//     Drive/Inputs/In/nDataIn1 <-> Inputs/Following error actual value
//     Drive/Inputs/In/nDcOutputTime <-> InfoData/DcOutputShift
//     Drive/Inputs/In/nState1 <-> Inputs/Statusword
//     Drive/Inputs/In/nState2 <-> Inputs/Statusword @bit 8
//     Drive/Inputs/In/nState4 @bit 1 <-> WcState/InputToggle
//     Drive/Inputs/In/nState4 <-> WcState/WcState
//     Drive/Outputs/Out/nCtrl1 <-> Outputs/Controlword
//     Drive/Outputs/Out/nCtrl2 <-> Outputs/Controlword @bit 8
//     Drive/Outputs/Out/nDataOut1 <-> Outputs/Target position
//     Enc/Inputs/In/nDataIn1 <-> Inputs/Position actual value
//     Enc/Inputs/In/nDataIn3 <-> Inputs/Touch probe pos1 pos value
//     Enc/Inputs/In/nDataIn5 <-> Inputs/Touch probe pos2 pos value
//     Enc/Inputs/In/nDcInputTime <-> InfoData/DcInputShift
//     Enc/Inputs/In/nState4 @bit 1 <-> WcState/InputToggle
//     Enc/Inputs/In/nState4 <-> WcState/WcState
//     Enc/Inputs/In/nState5 <-> Inputs/Touch probe status
//     Enc/Inputs/In/nState6 <-> Inputs/Touch probe status @bit 8
//     Enc/Outputs/Out/nCtrl5 <-> Outputs/Touch probe function
//     Enc/Outputs/Out/nCtrl6 <-> Outputs/Touch probe function @bit 8
//   NC-Task 1 SAF/Axes/Axis017_17 P1An_NGPush2 <-> Device 3 (EtherCAT)/Box 2 (CU1128)/正极踢单张废料(InoSV660N)
//     Drive/Inputs/In/nDataIn1 <-> Inputs/Following error actual value
//     Drive/Inputs/In/nDcOutputTime <-> InfoData/DcOutputShift
//     Drive/Inputs/In/nState1 <-> Inputs/Statusword
//     Drive/Inputs/In/nState2 <-> Inputs/Statusword @bit 8
//     Drive/Inputs/In/nState4 @bit 1 <-> WcState/InputToggle
//     Drive/Inputs/In/nState4 <-> WcState/WcState
//     Drive/Outputs/Out/nCtrl1 <-> Outputs/Controlword
//     Drive/Outputs/Out/nCtrl2 <-> Outputs/Controlword @bit 8
//     Drive/Outputs/Out/nDataOut1 <-> Outputs/Target position
//     Enc/Inputs/In/nDataIn1 <-> Inputs/Position actual value
//     Enc/Inputs/In/nDataIn3 <-> Inputs/Touch probe pos1 pos value
//     Enc/Inputs/In/nDataIn5 <-> Inputs/Touch probe pos2 pos value
//     Enc/Inputs/In/nDcInputTime <-> InfoData/DcInputShift
//     Enc/Inputs/In/nState4 @bit 1 <-> WcState/InputToggle
//     Enc/Inputs/In/nState4 <-> WcState/WcState
//     Enc/Inputs/In/nState5 <-> Inputs/Touch probe status
//     Enc/Inputs/In/nState6 <-> Inputs/Touch probe status @bit 8
//     Enc/Outputs/Out/nCtrl5 <-> Outputs/Touch probe function
//     Enc/Outputs/Out/nCtrl6 <-> Outputs/Touch probe function @bit 8
//   NC-Task 1 SAF/Axes/Axis018_18 P1An_DedustBelt <-> Device 3 (EtherCAT)/Box 2 (CU1128)/正极上表面除尘皮带(InoSV660N)
//     Drive/Inputs/In/nDataIn1 <-> Inputs/Following error actual value
//     Drive/Inputs/In/nDcOutputTime <-> InfoData/DcOutputShift
//     Drive/Inputs/In/nState1 <-> Inputs/Statusword
//     Drive/Inputs/In/nState2 <-> Inputs/Statusword @bit 8
//     Drive/Inputs/In/nState4 @bit 1 <-> WcState/InputToggle
//     Drive/Inputs/In/nState4 <-> WcState/WcState
//     Drive/Outputs/Out/nCtrl1 <-> Outputs/Controlword
//     Drive/Outputs/Out/nCtrl2 <-> Outputs/Controlword @bit 8
//     Drive/Outputs/Out/nDataOut1 <-> Outputs/Target position
//     Enc/Inputs/In/nDataIn1 <-> Inputs/Position actual value
//     Enc/Inputs/In/nDataIn3 <-> Inputs/Touch probe pos1 pos value
//     Enc/Inputs/In/nDataIn5 <-> Inputs/Touch probe pos2 pos value
//     Enc/Inputs/In/nDcInputTime <-> InfoData/DcInputShift
//     Enc/Inputs/In/nState4 @bit 1 <-> WcState/InputToggle
//     Enc/Inputs/In/nState4 <-> WcState/WcState
//     Enc/Inputs/In/nState5 <-> Inputs/Touch probe status
//     Enc/Inputs/In/nState6 <-> Inputs/Touch probe status @bit 8
//     Enc/Outputs/Out/nCtrl5 <-> Outputs/Touch probe function
//     Enc/Outputs/Out/nCtrl6 <-> Outputs/Touch probe function @bit 8
//   NC-Task 1 SAF/Axes/Axis019_19 P1An_DedustReverseBelt <-> Device 3 (EtherCAT)/Box 2 (CU1128)/正极下表面除尘倒装皮带(InoSV660N)
//     Drive/Inputs/In/nDataIn1 <-> Inputs/Following error actual value
//     Drive/Inputs/In/nDcOutputTime <-> InfoData/DcOutputShift
//     Drive/Inputs/In/nState1 <-> Inputs/Statusword
//     Drive/Inputs/In/nState2 <-> Inputs/Statusword @bit 8
//     Drive/Inputs/In/nState4 @bit 1 <-> WcState/InputToggle
//     Drive/Inputs/In/nState4 <-> WcState/WcState
//     Drive/Outputs/Out/nCtrl1 <-> Outputs/Controlword
//     Drive/Outputs/Out/nCtrl2 <-> Outputs/Controlword @bit 8
//     Drive/Outputs/Out/nDataOut1 <-> Outputs/Target position
//     Enc/Inputs/In/nDataIn1 <-> Inputs/Position actual value
//     Enc/Inputs/In/nDataIn3 <-> Inputs/Touch probe pos1 pos value
//     Enc/Inputs/In/nDataIn5 <-> Inputs/Touch probe pos2 pos value
//     Enc/Inputs/In/nDcInputTime <-> InfoData/DcInputShift
//     Enc/Inputs/In/nState4 @bit 1 <-> WcState/InputToggle
//     Enc/Inputs/In/nState4 <-> WcState/WcState
//     Enc/Inputs/In/nState5 <-> Inputs/Touch probe status
//     Enc/Inputs/In/nState6 <-> Inputs/Touch probe status @bit 8
//     Enc/Outputs/Out/nCtrl5 <-> Outputs/Touch probe function
//     Enc/Outputs/Out/nCtrl6 <-> Outputs/Touch probe function @bit 8
//   NC-Task 1 SAF/Axes/Axis020_20 P1An_SubBelt1 <-> Device 3 (EtherCAT)/P2M1正极送料分段皮带1[20(模切)] (InoSV660N)
//     Drive/Inputs/In/nDataIn1 <-> Inputs/Following error actual value
//     Drive/Inputs/In/nDcOutputTime <-> InfoData/DcOutputShift
//     Drive/Inputs/In/nState1 <-> Inputs/Statusword
//     Drive/Inputs/In/nState2 <-> Inputs/Statusword @bit 8
//     Drive/Inputs/In/nState4 @bit 1 <-> WcState/InputToggle
//     Drive/Inputs/In/nState4 <-> WcState/WcState
//     Drive/Outputs/Out/nCtrl1 <-> Outputs/Controlword
//     Drive/Outputs/Out/nCtrl2 <-> Outputs/Controlword @bit 8
//     Drive/Outputs/Out/nDataOut1 <-> Outputs/Target position
//     Enc/Inputs/In/nDataIn1 <-> Inputs/Position actual value
//     Enc/Inputs/In/nDataIn3 <-> Inputs/Touch probe pos1 pos value
//     Enc/Inputs/In/nDataIn5 <-> Inputs/Touch probe pos2 pos value
//     Enc/Inputs/In/nDcInputTime <-> InfoData/DcInputShift
//     Enc/Inputs/In/nState4 @bit 1 <-> WcState/InputToggle
//     Enc/Inputs/In/nState4 <-> WcState/WcState
//     Enc/Inputs/In/nState5 <-> Inputs/Touch probe status
//     Enc/Inputs/In/nState6 <-> Inputs/Touch probe status @bit 8
//     Enc/Outputs/Out/nCtrl5 <-> Outputs/Touch probe function
//     Enc/Outputs/Out/nCtrl6 <-> Outputs/Touch probe function @bit 8
//   NC-Task 1 SAF/Axes/Axis021_21 P1An_SubBelt2 <-> Device 3 (EtherCAT)/Box 2 (CU1128)/Term 44 (CU1128-C)/P2M2正极送料分段皮带2[21(模切)] (InoSV660N)
//     Drive/Inputs/In/nDataIn1 <-> Inputs/Following error actual value
//     Drive/Inputs/In/nDcOutputTime <-> InfoData/DcOutputShift
//     Drive/Inputs/In/nState1 <-> Inputs/Statusword
//     Drive/Inputs/In/nState2 <-> Inputs/Statusword @bit 8
//     Drive/Inputs/In/nState4 @bit 1 <-> WcState/InputToggle
//     Drive/Inputs/In/nState4 <-> WcState/WcState
//     Drive/Outputs/Out/nCtrl1 <-> Outputs/Controlword
//     Drive/Outputs/Out/nCtrl2 <-> Outputs/Controlword @bit 8
//     Drive/Outputs/Out/nDataOut1 <-> Outputs/Target position
//     Enc/Inputs/In/nDataIn1 <-> Inputs/Position actual value
//     Enc/Inputs/In/nDataIn3 <-> Inputs/Touch probe pos1 pos value
//     Enc/Inputs/In/nDataIn5 <-> Inputs/Touch probe pos2 pos value
//     Enc/Inputs/In/nDcInputTime <-> InfoData/DcInputShift
//     Enc/Inputs/In/nState4 @bit 1 <-> WcState/InputToggle
//     Enc/Inputs/In/nState4 <-> WcState/WcState
//     Enc/Inputs/In/nState5 <-> Inputs/Touch probe status
//     Enc/Inputs/In/nState6 <-> Inputs/Touch probe status @bit 8
//     Enc/Outputs/Out/nCtrl5 <-> Outputs/Touch probe function
//     Enc/Outputs/Out/nCtrl6 <-> Outputs/Touch probe function @bit 8
//   NC-Task 1 SAF/Axes/Axis022_22 P1An_SubBelt3 <-> Device 3 (EtherCAT)/Box 2 (CU1128)/Term 44 (CU1128-C)/P2M3正极送料分段皮带3（22模切） (InoSV660N)
//     Drive/Inputs/In/nDataIn1 <-> Inputs/Following error actual value
//     Drive/Inputs/In/nDcOutputTime <-> InfoData/DcOutputShift
//     Drive/Inputs/In/nState1 <-> Inputs/Statusword
//     Drive/Inputs/In/nState2 <-> Inputs/Statusword @bit 8
//     Drive/Inputs/In/nState4 @bit 1 <-> WcState/InputToggle
//     Drive/Inputs/In/nState4 <-> WcState/WcState
//     Drive/Outputs/Out/nCtrl1 <-> Outputs/Controlword
//     Drive/Outputs/Out/nCtrl2 <-> Outputs/Controlword @bit 8
//     Drive/Outputs/Out/nDataOut1 <-> Outputs/Target position
//     Enc/Inputs/In/nDataIn1 <-> Inputs/Position actual value
//     Enc/Inputs/In/nDataIn3 <-> Inputs/Touch probe pos1 pos value
//     Enc/Inputs/In/nDataIn5 <-> Inputs/Touch probe pos2 pos value
//     Enc/Inputs/In/nDcInputTime <-> InfoData/DcInputShift
//     Enc/Inputs/In/nState4 @bit 1 <-> WcState/InputToggle
//     Enc/Inputs/In/nState4 <-> WcState/WcState
//     Enc/Inputs/In/nState5 <-> Inputs/Touch probe status
//     Enc/Inputs/In/nState6 <-> Inputs/Touch probe status @bit 8
//     Enc/Outputs/Out/nCtrl5 <-> Outputs/Touch probe function
//     Enc/Outputs/Out/nCtrl6 <-> Outputs/Touch probe function @bit 8
//   NC-Task 1 SAF/Axes/Axis025_25 P1Ca_UnWind_L <-> Device 3 (EtherCAT)/Box 2 (CU1128)/Term 24 (CU1128-B)/负极左放卷电机(InoSV660N)
//     Drive/Inputs/In/nDataIn1 <-> Inputs/Following error actual value
//     Drive/Inputs/In/nDcOutputTime <-> InfoData/DcOutputShift
//     Drive/Inputs/In/nState1 <-> Inputs/Statusword
//     Drive/Inputs/In/nState2 <-> Inputs/Statusword @bit 8
//     Drive/Inputs/In/nState4 @bit 1 <-> WcState/InputToggle
//     Drive/Inputs/In/nState4 <-> WcState/WcState
//     Drive/Outputs/Out/nCtrl1 <-> Outputs/Controlword
//     Drive/Outputs/Out/nCtrl2 <-> Outputs/Controlword @bit 8
//     Drive/Outputs/Out/nDataOut1 <-> Outputs/Target position
//     Enc/Inputs/In/nDataIn1 <-> Inputs/Position actual value
//     Enc/Inputs/In/nDataIn3 <-> Inputs/Touch probe pos1 pos value
//     Enc/Inputs/In/nDataIn5 <-> Inputs/Touch probe pos2 pos value
//     Enc/Inputs/In/nDcInputTime <-> InfoData/DcInputShift
//     Enc/Inputs/In/nState4 @bit 1 <-> WcState/InputToggle
//     Enc/Inputs/In/nState4 <-> WcState/WcState
//     Enc/Inputs/In/nState5 <-> Inputs/Touch probe status
//     Enc/Inputs/In/nState6 <-> Inputs/Touch probe status @bit 8
//     Enc/Outputs/Out/nCtrl5 <-> Outputs/Touch probe function
//     Enc/Outputs/Out/nCtrl6 <-> Outputs/Touch probe function @bit 8
//   NC-Task 1 SAF/Axes/Axis026_26 P1Ca_UnWind_R <-> Device 3 (EtherCAT)/Box 2 (CU1128)/Term 24 (CU1128-B)/负极右放卷电机(InoSV660N)
//     Drive/Inputs/In/nDataIn1 <-> Inputs/Following error actual value
//     Drive/Inputs/In/nDcOutputTime <-> InfoData/DcOutputShift
//     Drive/Inputs/In/nState1 <-> Inputs/Statusword
//     Drive/Inputs/In/nState2 <-> Inputs/Statusword @bit 8
//     Drive/Inputs/In/nState4 @bit 1 <-> WcState/InputToggle
//     Drive/Inputs/In/nState4 <-> WcState/WcState
//     Drive/Outputs/Out/nCtrl1 <-> Outputs/Controlword
//     Drive/Outputs/Out/nCtrl2 <-> Outputs/Controlword @bit 8
//     Drive/Outputs/Out/nDataOut1 <-> Outputs/Target position
//     Enc/Inputs/In/nDataIn1 <-> Inputs/Position actual value
//     Enc/Inputs/In/nDataIn3 <-> Inputs/Touch probe pos1 pos value
//     Enc/Inputs/In/nDataIn5 <-> Inputs/Touch probe pos2 pos value
//     Enc/Inputs/In/nDcInputTime <-> InfoData/DcInputShift
//     Enc/Inputs/In/nState4 @bit 1 <-> WcState/InputToggle
//     Enc/Inputs/In/nState4 <-> WcState/WcState
//     Enc/Inputs/In/nState5 <-> Inputs/Touch probe status
//     Enc/Inputs/In/nState6 <-> Inputs/Touch probe status @bit 8
//     Enc/Outputs/Out/nCtrl5 <-> Outputs/Touch probe function
//     Enc/Outputs/Out/nCtrl6 <-> Outputs/Touch probe function @bit 8
//   NC-Task 1 SAF/Axes/Axis027_27 P1Ca_PoleTension <-> Device 3 (EtherCAT)/Box 2 (CU1128)/Term 24 (CU1128-B)/负极模切前摆杆张力(InoSV660N)
//     Drive/Inputs/In/nDcOutputTime <-> InfoData/DcOutputShift
//     Drive/Inputs/In/nState1 <-> Inputs/Statusword
//     Drive/Inputs/In/nState2 <-> Inputs/Statusword @bit 8
//     Drive/Inputs/In/nState4 @bit 1 <-> WcState/InputToggle
//     Drive/Inputs/In/nState4 <-> WcState/WcState
//     Drive/Inputs/In/nState5 <-> Inputs/Modes of operation display
//     Drive/Outputs/Out/nCtrl1 <-> Outputs/Controlword
//     Drive/Outputs/Out/nCtrl2 <-> Outputs/Controlword @bit 8
//     Drive/Outputs/Out/nDataOut1 <-> Outputs/Target position
//     Drive/Outputs/Out/nDataOut2 <-> Outputs/Target velocity
//     Enc/Inputs/In/nDataIn1 <-> Inputs/Position actual value
//     Enc/Inputs/In/nDataIn3 <-> Inputs/Touch probe pos1 pos value
//     Enc/Inputs/In/nDataIn5 <-> Inputs/Touch probe pos2 pos value
//     Enc/Inputs/In/nDcInputTime <-> InfoData/DcInputShift
//     Enc/Inputs/In/nState4 @bit 1 <-> WcState/InputToggle
//     Enc/Inputs/In/nState4 <-> WcState/WcState
//     Enc/Inputs/In/nState5 <-> Inputs/Touch probe status
//     Enc/Inputs/In/nState6 <-> Inputs/Touch probe status @bit 8
//     Enc/Outputs/Out/nCtrl5 <-> Outputs/Touch probe function
//     Enc/Outputs/Out/nCtrl6 <-> Outputs/Touch probe function @bit 8
//   NC-Task 1 SAF/Axes/Axis028_28 P1Ca_DriverAux <-> Device 3 (EtherCAT)/Box 2 (CU1128)/Term 24 (CU1128-B)/负极模切辅助驱动(InoSV660N)
//     Drive/Inputs/In/nDataIn1 <-> Inputs/Following error actual value
//     Drive/Inputs/In/nDcOutputTime <-> InfoData/DcOutputShift
//     Drive/Inputs/In/nState1 <-> Inputs/Statusword
//     Drive/Inputs/In/nState2 <-> Inputs/Statusword @bit 8
//     Drive/Inputs/In/nState4 @bit 1 <-> WcState/InputToggle
//     Drive/Inputs/In/nState4 <-> WcState/WcState
//     Drive/Outputs/Out/nCtrl1 <-> Outputs/Controlword
//     Drive/Outputs/Out/nCtrl2 <-> Outputs/Controlword @bit 8
//     Drive/Outputs/Out/nDataOut1 <-> Outputs/Target position
//     Enc/Inputs/In/nDataIn1 <-> Inputs/Position actual value
//     Enc/Inputs/In/nDataIn3 <-> Inputs/Touch probe pos1 pos value
//     Enc/Inputs/In/nDataIn5 <-> Inputs/Touch probe pos2 pos value
//     Enc/Inputs/In/nDcInputTime <-> InfoData/DcInputShift
//     Enc/Inputs/In/nState4 @bit 1 <-> WcState/InputToggle
//     Enc/Inputs/In/nState4 <-> WcState/WcState
//     Enc/Inputs/In/nState5 <-> Inputs/Touch probe status
//     Enc/Inputs/In/nState6 <-> Inputs/Touch probe status @bit 8
//     Enc/Outputs/Out/nCtrl5 <-> Outputs/Touch probe function
//     Enc/Outputs/Out/nCtrl6 <-> Outputs/Touch probe function @bit 8
//   NC-Task 1 SAF/Axes/Axis029_29 P1Ca_BuffeLine <-> Device 3 (EtherCAT)/Box 2 (CU1128)/Term 24 (CU1128-B)/负极模切极片缓存(CDHD)
//     Drive/Inputs/In/nDataIn1 <-> TxPDO 4/Following Error Actual Value
//     Drive/Inputs/In/nDcOutputTime <-> InfoData/DcOutputShift
//     Drive/Inputs/In/nState1 <-> TxPDO 1/StatusWord
//     Drive/Inputs/In/nState2 <-> TxPDO 1/StatusWord @bit 8
//     Drive/Inputs/In/nState4 @bit 1 <-> WcState/InputToggle
//     Drive/Inputs/In/nState4 <-> WcState/WcState
//     Drive/Inputs/In/nState5 <-> TxPDO 1/Modes of operation display
//     Drive/Outputs/Out/nCtrl1 <-> RxPDO 1/ControlWord
//     Drive/Outputs/Out/nCtrl2 <-> RxPDO 1/ControlWord @bit 8
//     Drive/Outputs/Out/nCtrl5 <-> RxPDO 1/Modes of operation
//     Drive/Outputs/Out/nDataOut1 <-> RxPDO 2/Target position
//     Drive/Outputs/Out/nDataOut2 <-> RxPDO 3/Target Velocity
//     Drive/Outputs/Out/nDataOut3[0] <-> RxPDO 4/Torque Offset
//     Drive/Outputs/Out/nDataOut4[0] <-> RxPDO 4/Target torque
//     Enc/Inputs/In/nDataIn1 <-> TxPDO 2/Position actual value
//     Enc/Inputs/In/nDcInputTime <-> InfoData/DcInputShift
//     Enc/Inputs/In/nState4 @bit 1 <-> WcState/InputToggle
//     Enc/Inputs/In/nState4 <-> WcState/WcState
//   NC-Task 1 SAF/Axes/Axis030_30 P1Ca_Mould <-> Device 3 (EtherCAT)/Box 2 (CU1128)/Term 24 (CU1128-B)/负极倒角模具(InoSV660N)
//     Drive/Inputs/In/nDataIn1 <-> Inputs/Following error actual value
//     Drive/Inputs/In/nDcOutputTime <-> InfoData/DcOutputShift
//     Drive/Inputs/In/nState1 <-> Inputs/Statusword
//     Drive/Inputs/In/nState2 <-> Inputs/Statusword @bit 8
//     Drive/Inputs/In/nState4 @bit 1 <-> WcState/InputToggle
//     Drive/Inputs/In/nState4 <-> WcState/WcState
//     Drive/Outputs/Out/nCtrl1 <-> Outputs/Controlword
//     Drive/Outputs/Out/nCtrl2 <-> Outputs/Controlword @bit 8
//     Drive/Outputs/Out/nDataOut1 <-> Outputs/Target position
//     Enc/Inputs/In/nDataIn1 <-> Inputs/Position actual value
//     Enc/Inputs/In/nDataIn3 <-> Inputs/Touch probe pos1 pos value
//     Enc/Inputs/In/nDataIn5 <-> Inputs/Touch probe pos2 pos value
//     Enc/Inputs/In/nDcInputTime <-> InfoData/DcInputShift
//     Enc/Inputs/In/nState4 @bit 1 <-> WcState/InputToggle
//     Enc/Inputs/In/nState4 <-> WcState/WcState
//     Enc/Inputs/In/nState5 <-> Inputs/Touch probe status
//     Enc/Inputs/In/nState6 <-> Inputs/Touch probe status @bit 8
//     Enc/Outputs/Out/nCtrl5 <-> Outputs/Touch probe function
//     Enc/Outputs/Out/nCtrl6 <-> Outputs/Touch probe function @bit 8
//   NC-Task 1 SAF/Axes/Axis031_31 P1Ca_MouldRectify_X <-> Device 3 (EtherCAT)/Box 2 (CU1128)/Term 24 (CU1128-B)/负极模具纠偏X轴(肩宽)(InoSV660N)
//     Drive/Inputs/In/nDataIn1 <-> Inputs/Following error actual value
//     Drive/Inputs/In/nDcOutputTime <-> InfoData/DcOutputShift
//     Drive/Inputs/In/nState1 <-> Inputs/Statusword
//     Drive/Inputs/In/nState2 <-> Inputs/Statusword @bit 8
//     Drive/Inputs/In/nState4 @bit 1 <-> WcState/InputToggle
//     Drive/Inputs/In/nState4 <-> WcState/WcState
//     Drive/Outputs/Out/nCtrl1 <-> Outputs/Controlword
//     Drive/Outputs/Out/nCtrl2 <-> Outputs/Controlword @bit 8
//     Drive/Outputs/Out/nDataOut1 <-> Outputs/Target position
//     Enc/Inputs/In/nDataIn1 <-> Inputs/Position actual value
//     Enc/Inputs/In/nDataIn3 <-> Inputs/Touch probe pos1 pos value
//     Enc/Inputs/In/nDataIn5 <-> Inputs/Touch probe pos2 pos value
//     Enc/Inputs/In/nDcInputTime <-> InfoData/DcInputShift
//     Enc/Inputs/In/nState4 @bit 1 <-> WcState/InputToggle
//     Enc/Inputs/In/nState4 <-> WcState/WcState
//     Enc/Inputs/In/nState5 <-> Inputs/Touch probe status
//     Enc/Inputs/In/nState6 <-> Inputs/Touch probe status @bit 8
//     Enc/Outputs/Out/nCtrl5 <-> Outputs/Touch probe function
//     Enc/Outputs/Out/nCtrl6 <-> Outputs/Touch probe function @bit 8
//   NC-Task 1 SAF/Axes/Axis032_32 P1Ca_MouldRectify_Y <-> Device 3 (EtherCAT)/Box 2 (CU1128)/Term 24 (CU1128-B)/负极模具纠偏Y轴(InoSV660N)
//     Drive/Inputs/In/nDataIn1 <-> Inputs/Following error actual value
//     Drive/Inputs/In/nDcOutputTime <-> InfoData/DcOutputShift
//     Drive/Inputs/In/nState1 <-> Inputs/Statusword
//     Drive/Inputs/In/nState2 <-> Inputs/Statusword @bit 8
//     Drive/Inputs/In/nState4 @bit 1 <-> WcState/InputToggle
//     Drive/Inputs/In/nState4 <-> WcState/WcState
//     Drive/Outputs/Out/nCtrl1 <-> Outputs/Controlword
//     Drive/Outputs/Out/nCtrl2 <-> Outputs/Controlword @bit 8
//     Drive/Outputs/Out/nDataOut1 <-> Outputs/Target position
//     Enc/Inputs/In/nDataIn1 <-> Inputs/Position actual value
//     Enc/Inputs/In/nDataIn3 <-> Inputs/Touch probe pos1 pos value
//     Enc/Inputs/In/nDataIn5 <-> Inputs/Touch probe pos2 pos value
//     Enc/Inputs/In/nDcInputTime <-> InfoData/DcInputShift
//     Enc/Inputs/In/nState4 @bit 1 <-> WcState/InputToggle
//     Enc/Inputs/In/nState4 <-> WcState/WcState
//     Enc/Inputs/In/nState5 <-> Inputs/Touch probe status
//     Enc/Inputs/In/nState6 <-> Inputs/Touch probe status @bit 8
//     Enc/Outputs/Out/nCtrl5 <-> Outputs/Touch probe function
//     Enc/Outputs/Out/nCtrl6 <-> Outputs/Touch probe function @bit 8
//   NC-Task 1 SAF/Axes/Axis033_33 P1Ca_DriverDDR <-> Device 3 (EtherCAT)/Box 2 (CU1128)/Term 24 (CU1128-B)/负极模切主驱动(CDHD)
//     Drive/Inputs/In/nDataIn1 <-> TxPDO 4/Following Error Actual Value
//     Drive/Inputs/In/nDcOutputTime <-> InfoData/DcOutputShift
//     Drive/Inputs/In/nState1 <-> TxPDO 1/StatusWord
//     Drive/Inputs/In/nState2 <-> TxPDO 1/StatusWord @bit 8
//     Drive/Inputs/In/nState4 @bit 1 <-> WcState/InputToggle
//     Drive/Inputs/In/nState4 <-> WcState/WcState
//     Drive/Inputs/In/nState5 <-> TxPDO 1/Modes of operation display
//     Drive/Outputs/Out/nCtrl1 <-> RxPDO 1/ControlWord
//     Drive/Outputs/Out/nCtrl2 <-> RxPDO 1/ControlWord @bit 8
//     Drive/Outputs/Out/nCtrl5 <-> RxPDO 1/Modes of operation
//     Drive/Outputs/Out/nDataOut1 <-> RxPDO 2/Target position
//     Drive/Outputs/Out/nDataOut2 <-> RxPDO 3/Target Velocity
//     Drive/Outputs/Out/nDataOut3[0] <-> RxPDO 4/Torque Offset
//     Drive/Outputs/Out/nDataOut4[0] <-> RxPDO 4/Target torque
//     Enc/Inputs/In/nDataIn1 <-> TxPDO 2/Position actual value
//     Enc/Inputs/In/nDcInputTime <-> InfoData/DcInputShift
//     Enc/Inputs/In/nState4 @bit 1 <-> WcState/InputToggle
//     Enc/Inputs/In/nState4 <-> WcState/WcState
//   NC-Task 1 SAF/Axes/Axis034_34 P1Ca_Cuter <-> Device 3 (EtherCAT)/Box 2 (CU1128)/Term 24 (CU1128-B)/负极裁切切刀(InoSV660N)
//     Drive/Inputs/In/nDataIn1 <-> Inputs/Following error actual value
//     Drive/Inputs/In/nDcOutputTime <-> InfoData/DcOutputShift
//     Drive/Inputs/In/nState1 <-> Inputs/Statusword
//     Drive/Inputs/In/nState2 <-> Inputs/Statusword @bit 8
//     Drive/Inputs/In/nState4 @bit 1 <-> WcState/InputToggle
//     Drive/Inputs/In/nState4 <-> WcState/WcState
//     Drive/Outputs/Out/nCtrl1 <-> Outputs/Controlword
//     Drive/Outputs/Out/nCtrl2 <-> Outputs/Controlword @bit 8
//     Drive/Outputs/Out/nDataOut1 <-> Outputs/Target position
//     Enc/Inputs/In/nDataIn1 <-> Inputs/Position actual value
//     Enc/Inputs/In/nDataIn3 <-> Inputs/Touch probe pos1 pos value
//     Enc/Inputs/In/nDataIn5 <-> Inputs/Touch probe pos2 pos value
//     Enc/Inputs/In/nDcInputTime <-> InfoData/DcInputShift
//     Enc/Inputs/In/nState4 @bit 1 <-> WcState/InputToggle
//     Enc/Inputs/In/nState4 <-> WcState/WcState
//     Enc/Inputs/In/nState5 <-> Inputs/Touch probe status
//     Enc/Inputs/In/nState6 <-> Inputs/Touch probe status @bit 8
//     Enc/Outputs/Out/nCtrl5 <-> Outputs/Touch probe function
//     Enc/Outputs/Out/nCtrl6 <-> Outputs/Touch probe function @bit 8
//   NC-Task 1 SAF/Axes/Axis035_35 P1Ca_CuterDegRectify <-> Device 3 (EtherCAT)/Box 2 (CU1128)/Term 24 (CU1128-B)/负极裁切角度纠偏(InoSV660N)
//     Drive/Inputs/In/nDataIn1 <-> Inputs/Following error actual value
//     Drive/Inputs/In/nDcOutputTime <-> InfoData/DcOutputShift
//     Drive/Inputs/In/nState1 <-> Inputs/Statusword
//     Drive/Inputs/In/nState2 <-> Inputs/Statusword @bit 8
//     Drive/Inputs/In/nState4 @bit 1 <-> WcState/InputToggle
//     Drive/Inputs/In/nState4 <-> WcState/WcState
//     Drive/Outputs/Out/nCtrl1 <-> Outputs/Controlword
//     Drive/Outputs/Out/nCtrl2 <-> Outputs/Controlword @bit 8
//     Drive/Outputs/Out/nDataOut1 <-> Outputs/Target position
//     Enc/Inputs/In/nDataIn1 <-> Inputs/Position actual value
//     Enc/Inputs/In/nDataIn3 <-> Inputs/Touch probe pos1 pos value
//     Enc/Inputs/In/nDataIn5 <-> Inputs/Touch probe pos2 pos value
//     Enc/Inputs/In/nDcInputTime <-> InfoData/DcInputShift
//     Enc/Inputs/In/nState4 @bit 1 <-> WcState/InputToggle
//     Enc/Inputs/In/nState4 <-> WcState/WcState
//     Enc/Inputs/In/nState5 <-> Inputs/Touch probe status
//     Enc/Inputs/In/nState6 <-> Inputs/Touch probe status @bit 8
//     Enc/Outputs/Out/nCtrl5 <-> Outputs/Touch probe function
//     Enc/Outputs/Out/nCtrl6 <-> Outputs/Touch probe function @bit 8
//   NC-Task 1 SAF/Axes/Axis036_36 P1Ca_CuterBelt <-> Device 3 (EtherCAT)/Box 2 (CU1128)/Term 24 (CU1128-B)/负极裁切输送皮带(InoSV660N)
//     Drive/Inputs/In/nDataIn1 <-> Inputs/Following error actual value
//     Drive/Inputs/In/nDcOutputTime <-> InfoData/DcOutputShift
//     Drive/Inputs/In/nState1 <-> Inputs/Statusword
//     Drive/Inputs/In/nState2 <-> Inputs/Statusword @bit 8
//     Drive/Inputs/In/nState4 @bit 1 <-> WcState/InputToggle
//     Drive/Inputs/In/nState4 <-> WcState/WcState
//     Drive/Outputs/Out/nCtrl1 <-> Outputs/Controlword
//     Drive/Outputs/Out/nCtrl2 <-> Outputs/Controlword @bit 8
//     Drive/Outputs/Out/nDataOut1 <-> Outputs/Target position
//     Enc/Inputs/In/nDataIn1 <-> Inputs/Position actual value
//     Enc/Inputs/In/nDataIn3 <-> Inputs/Touch probe pos1 pos value
//     Enc/Inputs/In/nDataIn5 <-> Inputs/Touch probe pos2 pos value
//     Enc/Inputs/In/nDcInputTime <-> InfoData/DcInputShift
//     Enc/Inputs/In/nState4 @bit 1 <-> WcState/InputToggle
//     Enc/Inputs/In/nState4 <-> WcState/WcState
//     Enc/Inputs/In/nState5 <-> Inputs/Touch probe status
//     Enc/Inputs/In/nState6 <-> Inputs/Touch probe status @bit 8
//     Enc/Outputs/Out/nCtrl5 <-> Outputs/Touch probe function
//     Enc/Outputs/Out/nCtrl6 <-> Outputs/Touch probe function @bit 8
//   NC-Task 1 SAF/Axes/Axis037_37 P1Ca_CuterBeltChange <-> Device 3 (EtherCAT)/Box 2 (CU1128)/Term 24 (CU1128-B)/负极裁切输送带换型(InoSV660N)
//     Drive/Inputs/In/nDataIn1 <-> Inputs/Following error actual value
//     Drive/Inputs/In/nDcOutputTime <-> InfoData/DcOutputShift
//     Drive/Inputs/In/nState1 <-> Inputs/Statusword
//     Drive/Inputs/In/nState2 <-> Inputs/Statusword @bit 8
//     Drive/Inputs/In/nState4 @bit 1 <-> WcState/InputToggle
//     Drive/Inputs/In/nState4 <-> WcState/WcState
//     Drive/Outputs/Out/nCtrl1 <-> Outputs/Controlword
//     Drive/Outputs/Out/nCtrl2 <-> Outputs/Controlword @bit 8
//     Drive/Outputs/Out/nDataOut1 <-> Outputs/Target position
//     Enc/Inputs/In/nDataIn1 <-> Inputs/Position actual value
//     Enc/Inputs/In/nDataIn3 <-> Inputs/Touch probe pos1 pos value
//     Enc/Inputs/In/nDataIn5 <-> Inputs/Touch probe pos2 pos value
//     Enc/Inputs/In/nDcInputTime <-> InfoData/DcInputShift
//     Enc/Inputs/In/nState4 @bit 1 <-> WcState/InputToggle
//     Enc/Inputs/In/nState4 <-> WcState/WcState
//     Enc/Inputs/In/nState5 <-> Inputs/Touch probe status
//     Enc/Inputs/In/nState6 <-> Inputs/Touch probe status @bit 8
//     Enc/Outputs/Out/nCtrl5 <-> Outputs/Touch probe function
//     Enc/Outputs/Out/nCtrl6 <-> Outputs/Touch probe function @bit 8
//   NC-Task 1 SAF/Axes/Axis038_38 P1Ca_CCDPressPush <-> Device 3 (EtherCAT)/Box 2 (CU1128)/Term 24 (CU1128-B)/负极尺寸CCD压片升降(InoSV660N)
//     Drive/Inputs/In/nDataIn1 <-> Inputs/Following error actual value
//     Drive/Inputs/In/nDcOutputTime <-> InfoData/DcOutputShift
//     Drive/Inputs/In/nState1 <-> Inputs/Statusword
//     Drive/Inputs/In/nState2 <-> Inputs/Statusword @bit 8
//     Drive/Inputs/In/nState4 @bit 1 <-> WcState/InputToggle
//     Drive/Inputs/In/nState4 <-> WcState/WcState
//     Drive/Outputs/Out/nCtrl1 <-> Outputs/Controlword
//     Drive/Outputs/Out/nCtrl2 <-> Outputs/Controlword @bit 8
//     Drive/Outputs/Out/nDataOut1 <-> Outputs/Target position
//     Enc/Inputs/In/nDataIn1 <-> Inputs/Position actual value
//     Enc/Inputs/In/nDataIn3 <-> Inputs/Touch probe pos1 pos value
//     Enc/Inputs/In/nDataIn5 <-> Inputs/Touch probe pos2 pos value
//     Enc/Inputs/In/nDcInputTime <-> InfoData/DcInputShift
//     Enc/Inputs/In/nState4 @bit 1 <-> WcState/InputToggle
//     Enc/Inputs/In/nState4 <-> WcState/WcState
//     Enc/Inputs/In/nState5 <-> Inputs/Touch probe status
//     Enc/Inputs/In/nState6 <-> Inputs/Touch probe status @bit 8
//     Enc/Outputs/Out/nCtrl5 <-> Outputs/Touch probe function
//     Enc/Outputs/Out/nCtrl6 <-> Outputs/Touch probe function @bit 8
//   NC-Task 1 SAF/Axes/Axis039_39 P1Ca_NGPushReverseBelt <-> Device 3 (EtherCAT)/Box 2 (CU1128)/Term 24 (CU1128-B)/负极踢废倒装皮带(InoSV660N)
//     Drive/Inputs/In/nDataIn1 <-> Inputs/Following error actual value
//     Drive/Inputs/In/nDcOutputTime <-> InfoData/DcOutputShift
//     Drive/Inputs/In/nState1 <-> Inputs/Statusword
//     Drive/Inputs/In/nState2 <-> Inputs/Statusword @bit 8
//     Drive/Inputs/In/nState4 @bit 1 <-> WcState/InputToggle
//     Drive/Inputs/In/nState4 <-> WcState/WcState
//     Drive/Outputs/Out/nCtrl1 <-> Outputs/Controlword
//     Drive/Outputs/Out/nCtrl2 <-> Outputs/Controlword @bit 8
//     Drive/Outputs/Out/nDataOut1 <-> Outputs/Target position
//     Enc/Inputs/In/nDataIn1 <-> Inputs/Position actual value
//     Enc/Inputs/In/nDataIn3 <-> Inputs/Touch probe pos1 pos value
//     Enc/Inputs/In/nDataIn5 <-> Inputs/Touch probe pos2 pos value
//     Enc/Inputs/In/nDcInputTime <-> InfoData/DcInputShift
//     Enc/Inputs/In/nState4 @bit 1 <-> WcState/InputToggle
//     Enc/Inputs/In/nState4 <-> WcState/WcState
//     Enc/Inputs/In/nState5 <-> Inputs/Touch probe status
//     Enc/Inputs/In/nState6 <-> Inputs/Touch probe status @bit 8
//     Enc/Outputs/Out/nCtrl5 <-> Outputs/Touch probe function
//     Enc/Outputs/Out/nCtrl6 <-> Outputs/Touch probe function @bit 8
//   NC-Task 1 SAF/Axes/Axis040_40 P1Ca_NGPush1 <-> Device 3 (EtherCAT)/Box 2 (CU1128)/Term 24 (CU1128-B)/负极踢连续废料(InoSV660N)
//     Drive/Inputs/In/nDataIn1 <-> Inputs/Following error actual value
//     Drive/Inputs/In/nDcOutputTime <-> InfoData/DcOutputShift
//     Drive/Inputs/In/nState1 <-> Inputs/Statusword
//     Drive/Inputs/In/nState2 <-> Inputs/Statusword @bit 8
//     Drive/Inputs/In/nState4 @bit 1 <-> WcState/InputToggle
//     Drive/Inputs/In/nState4 <-> WcState/WcState
//     Drive/Outputs/Out/nCtrl1 <-> Outputs/Controlword
//     Drive/Outputs/Out/nCtrl2 <-> Outputs/Controlword @bit 8
//     Drive/Outputs/Out/nDataOut1 <-> Outputs/Target position
//     Enc/Inputs/In/nDataIn1 <-> Inputs/Position actual value
//     Enc/Inputs/In/nDataIn3 <-> Inputs/Touch probe pos1 pos value
//     Enc/Inputs/In/nDataIn5 <-> Inputs/Touch probe pos2 pos value
//     Enc/Inputs/In/nDcInputTime <-> InfoData/DcInputShift
//     Enc/Inputs/In/nState4 @bit 1 <-> WcState/InputToggle
//     Enc/Inputs/In/nState4 <-> WcState/WcState
//     Enc/Inputs/In/nState5 <-> Inputs/Touch probe status
//     Enc/Inputs/In/nState6 <-> Inputs/Touch probe status @bit 8
//     Enc/Outputs/Out/nCtrl5 <-> Outputs/Touch probe function
//     Enc/Outputs/Out/nCtrl6 <-> Outputs/Touch probe function @bit 8
//   NC-Task 1 SAF/Axes/Axis041_41 P1Ca_NGPush2 <-> Device 3 (EtherCAT)/Box 2 (CU1128)/Term 24 (CU1128-B)/负极踢单张废料(InoSV660N)
//     Drive/Inputs/In/nDataIn1 <-> Inputs/Following error actual value
//     Drive/Inputs/In/nDcOutputTime <-> InfoData/DcOutputShift
//     Drive/Inputs/In/nState1 <-> Inputs/Statusword
//     Drive/Inputs/In/nState2 <-> Inputs/Statusword @bit 8
//     Drive/Inputs/In/nState4 @bit 1 <-> WcState/InputToggle
//     Drive/Inputs/In/nState4 <-> WcState/WcState
//     Drive/Outputs/Out/nCtrl1 <-> Outputs/Controlword
//     Drive/Outputs/Out/nCtrl2 <-> Outputs/Controlword @bit 8
//     Drive/Outputs/Out/nDataOut1 <-> Outputs/Target position
//     Enc/Inputs/In/nDataIn1 <-> Inputs/Position actual value
//     Enc/Inputs/In/nDataIn3 <-> Inputs/Touch probe pos1 pos value
//     Enc/Inputs/In/nDataIn5 <-> Inputs/Touch probe pos2 pos value
//     Enc/Inputs/In/nDcInputTime <-> InfoData/DcInputShift
//     Enc/Inputs/In/nState4 @bit 1 <-> WcState/InputToggle
//     Enc/Inputs/In/nState4 <-> WcState/WcState
//     Enc/Inputs/In/nState5 <-> Inputs/Touch probe status
//     Enc/Inputs/In/nState6 <-> Inputs/Touch probe status @bit 8
//     Enc/Outputs/Out/nCtrl5 <-> Outputs/Touch probe function
//     Enc/Outputs/Out/nCtrl6 <-> Outputs/Touch probe function @bit 8
//   NC-Task 1 SAF/Axes/Axis042_42 P1Ca_DedustBelt <-> Device 3 (EtherCAT)/Box 2 (CU1128)/Term 24 (CU1128-B)/负极上表面除尘皮带(InoSV660N)
//     Drive/Inputs/In/nDataIn1 <-> Inputs/Following error actual value
//     Drive/Inputs/In/nDcOutputTime <-> InfoData/DcOutputShift
//     Drive/Inputs/In/nState1 <-> Inputs/Statusword
//     Drive/Inputs/In/nState2 <-> Inputs/Statusword @bit 8
//     Drive/Inputs/In/nState4 @bit 1 <-> WcState/InputToggle
//     Drive/Inputs/In/nState4 <-> WcState/WcState
//     Drive/Outputs/Out/nCtrl1 <-> Outputs/Controlword
//     Drive/Outputs/Out/nCtrl2 <-> Outputs/Controlword @bit 8
//     Drive/Outputs/Out/nDataOut1 <-> Outputs/Target position
//     Enc/Inputs/In/nDataIn1 <-> Inputs/Position actual value
//     Enc/Inputs/In/nDataIn3 <-> Inputs/Touch probe pos1 pos value
//     Enc/Inputs/In/nDataIn5 <-> Inputs/Touch probe pos2 pos value
//     Enc/Inputs/In/nDcInputTime <-> InfoData/DcInputShift
//     Enc/Inputs/In/nState4 @bit 1 <-> WcState/InputToggle
//     Enc/Inputs/In/nState4 <-> WcState/WcState
//     Enc/Inputs/In/nState5 <-> Inputs/Touch probe status
//     Enc/Inputs/In/nState6 <-> Inputs/Touch probe status @bit 8
//     Enc/Outputs/Out/nCtrl5 <-> Outputs/Touch probe function
//     Enc/Outputs/Out/nCtrl6 <-> Outputs/Touch probe function @bit 8
//   NC-Task 1 SAF/Axes/Axis043_43 P1Ca_DedustReverseBelt <-> Device 3 (EtherCAT)/Box 2 (CU1128)/Term 24 (CU1128-B)/负极下表面除尘倒装皮带(InoSV660N)
//     Drive/Inputs/In/nDataIn1 <-> Inputs/Following error actual value
//     Drive/Inputs/In/nDcOutputTime <-> InfoData/DcOutputShift
//     Drive/Inputs/In/nState1 <-> Inputs/Statusword
//     Drive/Inputs/In/nState2 <-> Inputs/Statusword @bit 8
//     Drive/Inputs/In/nState4 @bit 1 <-> WcState/InputToggle
//     Drive/Inputs/In/nState4 <-> WcState/WcState
//     Drive/Outputs/Out/nCtrl1 <-> Outputs/Controlword
//     Drive/Outputs/Out/nCtrl2 <-> Outputs/Controlword @bit 8
//     Drive/Outputs/Out/nDataOut1 <-> Outputs/Target position
//     Enc/Inputs/In/nDataIn1 <-> Inputs/Position actual value
//     Enc/Inputs/In/nDataIn3 <-> Inputs/Touch probe pos1 pos value
//     Enc/Inputs/In/nDataIn5 <-> Inputs/Touch probe pos2 pos value
//     Enc/Inputs/In/nDcInputTime <-> InfoData/DcInputShift
//     Enc/Inputs/In/nState4 @bit 1 <-> WcState/InputToggle
//     Enc/Inputs/In/nState4 <-> WcState/WcState
//     Enc/Inputs/In/nState5 <-> Inputs/Touch probe status
//     Enc/Inputs/In/nState6 <-> Inputs/Touch probe status @bit 8
//     Enc/Outputs/Out/nCtrl5 <-> Outputs/Touch probe function
//     Enc/Outputs/Out/nCtrl6 <-> Outputs/Touch probe function @bit 8
//   NC-Task 1 SAF/Axes/Axis044_44 P1Ca_SubBelt1 <-> Device 3 (EtherCAT)/P2M1负极送料分段皮带1[44（模切）] (InoSV660N)
//     Drive/Inputs/In/nDataIn1 <-> Inputs/Following error actual value
//     Drive/Inputs/In/nDcOutputTime <-> InfoData/DcOutputShift
//     Drive/Inputs/In/nState1 <-> Inputs/Statusword
//     Drive/Inputs/In/nState2 <-> Inputs/Statusword @bit 8
//     Drive/Inputs/In/nState4 @bit 1 <-> WcState/InputToggle
//     Drive/Inputs/In/nState4 <-> WcState/WcState
//     Drive/Outputs/Out/nCtrl1 <-> Outputs/Controlword
//     Drive/Outputs/Out/nCtrl2 <-> Outputs/Controlword @bit 8
//     Drive/Outputs/Out/nDataOut1 <-> Outputs/Target position
//     Enc/Inputs/In/nDataIn1 <-> Inputs/Position actual value
//     Enc/Inputs/In/nDataIn3 <-> Inputs/Touch probe pos1 pos value
//     Enc/Inputs/In/nDataIn5 <-> Inputs/Touch probe pos2 pos value
//     Enc/Inputs/In/nDcInputTime <-> InfoData/DcInputShift
//     Enc/Inputs/In/nState4 @bit 1 <-> WcState/InputToggle
//     Enc/Inputs/In/nState4 <-> WcState/WcState
//     Enc/Inputs/In/nState5 <-> Inputs/Touch probe status
//     Enc/Inputs/In/nState6 <-> Inputs/Touch probe status @bit 8
//     Enc/Outputs/Out/nCtrl5 <-> Outputs/Touch probe function
//     Enc/Outputs/Out/nCtrl6 <-> Outputs/Touch probe function @bit 8
//   NC-Task 1 SAF/Axes/Axis045_45 P1Ca_SubBelt2 <-> Device 3 (EtherCAT)/Box 2 (CU1128)/Term 44 (CU1128-C)/P2M2负极送料分段皮带2（45模切） (InoSV660N)
//     Drive/Inputs/In/nDataIn1 <-> Inputs/Following error actual value
//     Drive/Inputs/In/nDcOutputTime <-> InfoData/DcOutputShift
//     Drive/Inputs/In/nState1 <-> Inputs/Statusword
//     Drive/Inputs/In/nState2 <-> Inputs/Statusword @bit 8
//     Drive/Inputs/In/nState4 @bit 1 <-> WcState/InputToggle
//     Drive/Inputs/In/nState4 <-> WcState/WcState
//     Drive/Outputs/Out/nCtrl1 <-> Outputs/Controlword
//     Drive/Outputs/Out/nCtrl2 <-> Outputs/Controlword @bit 8
//     Drive/Outputs/Out/nDataOut1 <-> Outputs/Target position
//     Enc/Inputs/In/nDataIn1 <-> Inputs/Position actual value
//     Enc/Inputs/In/nDataIn3 <-> Inputs/Touch probe pos1 pos value
//     Enc/Inputs/In/nDataIn5 <-> Inputs/Touch probe pos2 pos value
//     Enc/Inputs/In/nDcInputTime <-> InfoData/DcInputShift
//     Enc/Inputs/In/nState4 @bit 1 <-> WcState/InputToggle
//     Enc/Inputs/In/nState4 <-> WcState/WcState
//     Enc/Inputs/In/nState5 <-> Inputs/Touch probe status
//     Enc/Inputs/In/nState6 <-> Inputs/Touch probe status @bit 8
//     Enc/Outputs/Out/nCtrl5 <-> Outputs/Touch probe function
//     Enc/Outputs/Out/nCtrl6 <-> Outputs/Touch probe function @bit 8
//   NC-Task 1 SAF/Axes/Axis046_46 P1Ca_SubBelt3 <-> Device 3 (EtherCAT)/Box 2 (CU1128)/Term 44 (CU1128-C)/P2M3负极送料分段皮带3（46模切） (InoSV660N)
//     Drive/Inputs/In/nDataIn1 <-> Inputs/Following error actual value
//     Drive/Inputs/In/nDcOutputTime <-> InfoData/DcOutputShift
//     Drive/Inputs/In/nState1 <-> Inputs/Statusword
//     Drive/Inputs/In/nState2 <-> Inputs/Statusword @bit 8
//     Drive/Inputs/In/nState4 @bit 1 <-> WcState/InputToggle
//     Drive/Inputs/In/nState4 <-> WcState/WcState
//     Drive/Outputs/Out/nCtrl1 <-> Outputs/Controlword
//     Drive/Outputs/Out/nCtrl2 <-> Outputs/Controlword @bit 8
//     Drive/Outputs/Out/nDataOut1 <-> Outputs/Target position
//     Enc/Inputs/In/nDataIn1 <-> Inputs/Position actual value
//     Enc/Inputs/In/nDataIn3 <-> Inputs/Touch probe pos1 pos value
//     Enc/Inputs/In/nDataIn5 <-> Inputs/Touch probe pos2 pos value
//     Enc/Inputs/In/nDcInputTime <-> InfoData/DcInputShift
//     Enc/Inputs/In/nState4 @bit 1 <-> WcState/InputToggle
//     Enc/Inputs/In/nState4 <-> WcState/WcState
//     Enc/Inputs/In/nState5 <-> Inputs/Touch probe status
//     Enc/Inputs/In/nState6 <-> Inputs/Touch probe status @bit 8
//     Enc/Outputs/Out/nCtrl5 <-> Outputs/Touch probe function
//     Enc/Outputs/Out/nCtrl6 <-> Outputs/Touch probe function @bit 8
//   NC-Task 1 SAF/Axes/Axis049_1 P2M1_AnCarryingLine <-> Device 3 (EtherCAT)/P2M1正极送片搬运平移[1](CDHD)
//     Drive/Inputs/In/nDataIn1 <-> TxPDO 4/Following Error Actual Value
//     Drive/Inputs/In/nDcOutputTime <-> InfoData/DcOutputShift
//     Drive/Inputs/In/nState1 <-> TxPDO 1/StatusWord
//     Drive/Inputs/In/nState2 <-> TxPDO 1/StatusWord @bit 8
//     Drive/Inputs/In/nState4 @bit 1 <-> WcState/InputToggle
//     Drive/Inputs/In/nState4 <-> WcState/WcState
//     Drive/Inputs/In/nState5 <-> TxPDO 1/Modes of operation display
//     Drive/Outputs/Out/nCtrl1 <-> RxPDO 1/ControlWord
//     Drive/Outputs/Out/nCtrl2 <-> RxPDO 1/ControlWord @bit 8
//     Drive/Outputs/Out/nCtrl5 <-> RxPDO 1/Modes of operation
//     Drive/Outputs/Out/nDataOut1 <-> RxPDO 2/Target position
//     Drive/Outputs/Out/nDataOut2 <-> RxPDO 3/Target Velocity
//     Drive/Outputs/Out/nDataOut3[0] <-> RxPDO 4/Torque Offset
//     Drive/Outputs/Out/nDataOut4[0] <-> RxPDO 4/Target torque
//     Enc/Inputs/In/nDataIn1 <-> TxPDO 2/Position actual value
//     Enc/Inputs/In/nDcInputTime <-> InfoData/DcInputShift
//     Enc/Inputs/In/nState4 @bit 1 <-> WcState/InputToggle
//     Enc/Inputs/In/nState4 <-> WcState/WcState
//   NC-Task 1 SAF/Axes/Axis050_2 P2M1_AnCarryingUpDown <-> Device 3 (EtherCAT)/P2M1正极送片搬运升降_[2] (InoSV660N)
//     Drive/Inputs/In/nDataIn1 <-> Inputs/Following error actual value
//     Drive/Inputs/In/nDcOutputTime <-> InfoData/DcOutputShift
//     Drive/Inputs/In/nState1 <-> Inputs/Statusword
//     Drive/Inputs/In/nState2 <-> Inputs/Statusword @bit 8
//     Drive/Inputs/In/nState4 @bit 1 <-> WcState/InputToggle
//     Drive/Inputs/In/nState4 <-> WcState/WcState
//     Drive/Outputs/Out/nCtrl1 <-> Outputs/Controlword
//     Drive/Outputs/Out/nCtrl2 <-> Outputs/Controlword @bit 8
//     Drive/Outputs/Out/nDataOut1 <-> Outputs/Target position
//     Enc/Inputs/In/nDataIn1 <-> Inputs/Position actual value
//     Enc/Inputs/In/nDataIn3 <-> Inputs/Touch probe pos1 pos value
//     Enc/Inputs/In/nDataIn5 <-> Inputs/Touch probe pos2 pos value
//     Enc/Inputs/In/nDcInputTime <-> InfoData/DcInputShift
//     Enc/Inputs/In/nState4 @bit 1 <-> WcState/InputToggle
//     Enc/Inputs/In/nState4 <-> WcState/WcState
//     Enc/Inputs/In/nState5 <-> Inputs/Touch probe status
//     Enc/Inputs/In/nState6 <-> Inputs/Touch probe status @bit 8
//     Enc/Outputs/Out/nCtrl5 <-> Outputs/Touch probe function
//     Enc/Outputs/Out/nCtrl6 <-> Outputs/Touch probe function @bit 8
//   NC-Task 1 SAF/Axes/Axis051_3 P2M1_AnCarryingWhirling <-> Device 3 (EtherCAT)/P2M1正极送片搬运旋转_3 (InoSV660N)
//     Drive/Inputs/In/nDataIn1 <-> Inputs/Following error actual value
//     Drive/Inputs/In/nDcOutputTime <-> InfoData/DcOutputShift
//     Drive/Inputs/In/nState1 <-> Inputs/Statusword
//     Drive/Inputs/In/nState2 <-> Inputs/Statusword @bit 8
//     Drive/Inputs/In/nState4 @bit 1 <-> WcState/InputToggle
//     Drive/Inputs/In/nState4 <-> WcState/WcState
//     Drive/Outputs/Out/nCtrl1 <-> Outputs/Controlword
//     Drive/Outputs/Out/nCtrl2 <-> Outputs/Controlword @bit 8
//     Drive/Outputs/Out/nDataOut1 <-> Outputs/Target position
//     Enc/Inputs/In/nDataIn1 <-> Inputs/Position actual value
//     Enc/Inputs/In/nDataIn3 <-> Inputs/Touch probe pos1 pos value
//     Enc/Inputs/In/nDataIn5 <-> Inputs/Touch probe pos2 pos value
//     Enc/Inputs/In/nDcInputTime <-> InfoData/DcInputShift
//     Enc/Inputs/In/nState4 @bit 1 <-> WcState/InputToggle
//     Enc/Inputs/In/nState4 <-> WcState/WcState
//     Enc/Inputs/In/nState5 <-> Inputs/Touch probe status
//     Enc/Inputs/In/nState6 <-> Inputs/Touch probe status @bit 8
//     Enc/Outputs/Out/nCtrl5 <-> Outputs/Touch probe function
//     Enc/Outputs/Out/nCtrl6 <-> Outputs/Touch probe function @bit 8
//   NC-Task 1 SAF/Axes/Axis052_4 P2M1_AnDTCarryingLine <-> Device 3 (EtherCAT)/P2M1正极叠台搬运平移1[4](CDHD)
//     Drive/Inputs/In/nDataIn1 <-> TxPDO 4/Following Error Actual Value
//     Drive/Inputs/In/nDcOutputTime <-> InfoData/DcOutputShift
//     Drive/Inputs/In/nState1 <-> TxPDO 1/StatusWord
//     Drive/Inputs/In/nState2 <-> TxPDO 1/StatusWord @bit 8
//     Drive/Inputs/In/nState4 @bit 1 <-> WcState/InputToggle
//     Drive/Inputs/In/nState4 <-> WcState/WcState
//     Drive/Inputs/In/nState5 <-> TxPDO 1/Modes of operation display
//     Drive/Outputs/Out/nCtrl1 <-> RxPDO 1/ControlWord
//     Drive/Outputs/Out/nCtrl2 <-> RxPDO 1/ControlWord @bit 8
//     Drive/Outputs/Out/nCtrl5 <-> RxPDO 1/Modes of operation
//     Drive/Outputs/Out/nDataOut1 <-> RxPDO 2/Target position
//     Drive/Outputs/Out/nDataOut2 <-> RxPDO 3/Target Velocity
//     Drive/Outputs/Out/nDataOut3[0] <-> RxPDO 4/Torque Offset
//     Drive/Outputs/Out/nDataOut4[0] <-> RxPDO 4/Target torque
//     Enc/Inputs/In/nDataIn1 <-> TxPDO 2/Position actual value
//     Enc/Inputs/In/nDcInputTime <-> InfoData/DcInputShift
//     Enc/Inputs/In/nState4 @bit 1 <-> WcState/InputToggle
//     Enc/Inputs/In/nState4 <-> WcState/WcState
//   NC-Task 1 SAF/Axes/Axis053_5 P2M1_AnDTCarryingUpDown <-> Device 3 (EtherCAT)/P2M1正极叠台搬运升降[5](InoSV660N)
//     Drive/Inputs/In/nDataIn1 <-> Inputs/Following error actual value
//     Drive/Inputs/In/nDcOutputTime <-> InfoData/DcOutputShift
//     Drive/Inputs/In/nState1 <-> Inputs/Statusword
//     Drive/Inputs/In/nState2 <-> Inputs/Statusword @bit 8
//     Drive/Inputs/In/nState4 @bit 1 <-> WcState/InputToggle
//     Drive/Inputs/In/nState4 <-> WcState/WcState
//     Drive/Outputs/Out/nCtrl1 <-> Outputs/Controlword
//     Drive/Outputs/Out/nCtrl2 <-> Outputs/Controlword @bit 8
//     Drive/Outputs/Out/nDataOut1 <-> Outputs/Target position
//     Enc/Inputs/In/nDataIn1 <-> Inputs/Position actual value
//     Enc/Inputs/In/nDataIn3 <-> Inputs/Touch probe pos1 pos value
//     Enc/Inputs/In/nDataIn5 <-> Inputs/Touch probe pos2 pos value
//     Enc/Inputs/In/nDcInputTime <-> InfoData/DcInputShift
//     Enc/Inputs/In/nState4 @bit 1 <-> WcState/InputToggle
//     Enc/Inputs/In/nState4 <-> WcState/WcState
//     Enc/Inputs/In/nState5 <-> Inputs/Touch probe status
//     Enc/Inputs/In/nState6 <-> Inputs/Touch probe status @bit 8
//     Enc/Outputs/Out/nCtrl5 <-> Outputs/Touch probe function
//     Enc/Outputs/Out/nCtrl6 <-> Outputs/Touch probe function @bit 8
//   NC-Task 1 SAF/Axes/Axis054_6 P2M1_AndeviationX1 <-> Device 3 (EtherCAT)/P2M1正极纠偏平台X1[6](InoSV660N)
//     Drive/Inputs/In/nDataIn1 <-> Inputs/Following error actual value
//     Drive/Inputs/In/nDcOutputTime <-> InfoData/DcOutputShift
//     Drive/Inputs/In/nState1 <-> Inputs/Statusword
//     Drive/Inputs/In/nState2 <-> Inputs/Statusword @bit 8
//     Drive/Inputs/In/nState4 @bit 1 <-> WcState/InputToggle
//     Drive/Inputs/In/nState4 <-> WcState/WcState
//     Drive/Outputs/Out/nCtrl1 <-> Outputs/Controlword
//     Drive/Outputs/Out/nCtrl2 <-> Outputs/Controlword @bit 8
//     Drive/Outputs/Out/nDataOut1 <-> Outputs/Target position
//     Enc/Inputs/In/nDataIn1 <-> Inputs/Position actual value
//     Enc/Inputs/In/nDataIn3 <-> Inputs/Touch probe pos1 pos value
//     Enc/Inputs/In/nDataIn5 <-> Inputs/Touch probe pos2 pos value
//     Enc/Inputs/In/nDcInputTime <-> InfoData/DcInputShift
//     Enc/Inputs/In/nState4 @bit 1 <-> WcState/InputToggle
//     Enc/Inputs/In/nState4 <-> WcState/WcState
//     Enc/Inputs/In/nState5 <-> Inputs/Touch probe status
//     Enc/Inputs/In/nState6 <-> Inputs/Touch probe status @bit 8
//     Enc/Outputs/Out/nCtrl5 <-> Outputs/Touch probe function
//     Enc/Outputs/Out/nCtrl6 <-> Outputs/Touch probe function @bit 8
//   NC-Task 1 SAF/Axes/Axis055_7 P2M1_AndeviationX2 <-> Device 3 (EtherCAT)/P2M1正极纠偏平台X2 [7](InoSV660N)
//     Drive/Inputs/In/nDataIn1 <-> Inputs/Following error actual value
//     Drive/Inputs/In/nDcOutputTime <-> InfoData/DcOutputShift
//     Drive/Inputs/In/nState1 <-> Inputs/Statusword
//     Drive/Inputs/In/nState2 <-> Inputs/Statusword @bit 8
//     Drive/Inputs/In/nState4 @bit 1 <-> WcState/InputToggle
//     Drive/Inputs/In/nState4 <-> WcState/WcState
//     Drive/Outputs/Out/nCtrl1 <-> Outputs/Controlword
//     Drive/Outputs/Out/nCtrl2 <-> Outputs/Controlword @bit 8
//     Drive/Outputs/Out/nDataOut1 <-> Outputs/Target position
//     Enc/Inputs/In/nDataIn1 <-> Inputs/Position actual value
//     Enc/Inputs/In/nDataIn3 <-> Inputs/Touch probe pos1 pos value
//     Enc/Inputs/In/nDataIn5 <-> Inputs/Touch probe pos2 pos value
//     Enc/Inputs/In/nDcInputTime <-> InfoData/DcInputShift
//     Enc/Inputs/In/nState4 @bit 1 <-> WcState/InputToggle
//     Enc/Inputs/In/nState4 <-> WcState/WcState
//     Enc/Inputs/In/nState5 <-> Inputs/Touch probe status
//     Enc/Inputs/In/nState6 <-> Inputs/Touch probe status @bit 8
//     Enc/Outputs/Out/nCtrl5 <-> Outputs/Touch probe function
//     Enc/Outputs/Out/nCtrl6 <-> Outputs/Touch probe function @bit 8
//   NC-Task 1 SAF/Axes/Axis056_8 P2M1_AndeviationY <-> Device 3 (EtherCAT)/P2M1正极纠偏平台Y [8](InoSV660N)
//     Drive/Inputs/In/nDataIn1 <-> Inputs/Following error actual value
//     Drive/Inputs/In/nDcOutputTime <-> InfoData/DcOutputShift
//     Drive/Inputs/In/nState1 <-> Inputs/Statusword
//     Drive/Inputs/In/nState2 <-> Inputs/Statusword @bit 8
//     Drive/Inputs/In/nState4 @bit 1 <-> WcState/InputToggle
//     Drive/Inputs/In/nState4 <-> WcState/WcState
//     Drive/Outputs/Out/nCtrl1 <-> Outputs/Controlword
//     Drive/Outputs/Out/nCtrl2 <-> Outputs/Controlword @bit 8
//     Drive/Outputs/Out/nDataOut1 <-> Outputs/Target position
//     Enc/Inputs/In/nDataIn1 <-> Inputs/Position actual value
//     Enc/Inputs/In/nDataIn3 <-> Inputs/Touch probe pos1 pos value
//     Enc/Inputs/In/nDataIn5 <-> Inputs/Touch probe pos2 pos value
//     Enc/Inputs/In/nDcInputTime <-> InfoData/DcInputShift
//     Enc/Inputs/In/nState4 @bit 1 <-> WcState/InputToggle
//     Enc/Inputs/In/nState4 <-> WcState/WcState
//     Enc/Inputs/In/nState5 <-> Inputs/Touch probe status
//     Enc/Inputs/In/nState6 <-> Inputs/Touch probe status @bit 8
//     Enc/Outputs/Out/nCtrl5 <-> Outputs/Touch probe function
//     Enc/Outputs/Out/nCtrl6 <-> Outputs/Touch probe function @bit 8
//   NC-Task 1 SAF/Axes/Axis057_9 P2M1_CaCarryingLine1 <-> Device 3 (EtherCAT)/P2M1负极送片搬运1平移[9](CDHD)
//     Drive/Inputs/In/nDataIn1 <-> TxPDO 4/Following Error Actual Value
//     Drive/Inputs/In/nDcOutputTime <-> InfoData/DcOutputShift
//     Drive/Inputs/In/nState1 <-> TxPDO 1/StatusWord
//     Drive/Inputs/In/nState2 <-> TxPDO 1/StatusWord @bit 8
//     Drive/Inputs/In/nState4 @bit 1 <-> WcState/InputToggle
//     Drive/Inputs/In/nState4 <-> WcState/WcState
//     Drive/Inputs/In/nState5 <-> TxPDO 1/Modes of operation display
//     Drive/Outputs/Out/nCtrl1 <-> RxPDO 1/ControlWord
//     Drive/Outputs/Out/nCtrl2 <-> RxPDO 1/ControlWord @bit 8
//     Drive/Outputs/Out/nCtrl5 <-> RxPDO 1/Modes of operation
//     Drive/Outputs/Out/nDataOut1 <-> RxPDO 2/Target position
//     Drive/Outputs/Out/nDataOut2 <-> RxPDO 3/Target Velocity
//     Drive/Outputs/Out/nDataOut3[0] <-> RxPDO 4/Torque Offset
//     Drive/Outputs/Out/nDataOut4[0] <-> RxPDO 4/Target torque
//     Enc/Inputs/In/nDataIn1 <-> TxPDO 2/Position actual value
//     Enc/Inputs/In/nDcInputTime <-> InfoData/DcInputShift
//     Enc/Inputs/In/nState4 @bit 1 <-> WcState/InputToggle
//     Enc/Inputs/In/nState4 <-> WcState/WcState
//   NC-Task 1 SAF/Axes/Axis058_10 P2M1_CaCarryingUpDown1 <-> Device 3 (EtherCAT)/P2M1负极送片搬运1升降[10] (InoSV660N)
//     Drive/Inputs/In/nDataIn1 <-> Inputs/Following error actual value
//     Drive/Inputs/In/nDcOutputTime <-> InfoData/DcOutputShift
//     Drive/Inputs/In/nState1 <-> Inputs/Statusword
//     Drive/Inputs/In/nState2 <-> Inputs/Statusword @bit 8
//     Drive/Inputs/In/nState4 @bit 1 <-> WcState/InputToggle
//     Drive/Inputs/In/nState4 <-> WcState/WcState
//     Drive/Outputs/Out/nCtrl1 <-> Outputs/Controlword
//     Drive/Outputs/Out/nCtrl2 <-> Outputs/Controlword @bit 8
//     Drive/Outputs/Out/nDataOut1 <-> Outputs/Target position
//     Enc/Inputs/In/nDataIn1 <-> Inputs/Position actual value
//     Enc/Inputs/In/nDataIn3 <-> Inputs/Touch probe pos1 pos value
//     Enc/Inputs/In/nDataIn5 <-> Inputs/Touch probe pos2 pos value
//     Enc/Inputs/In/nDcInputTime <-> InfoData/DcInputShift
//     Enc/Inputs/In/nState4 @bit 1 <-> WcState/InputToggle
//     Enc/Inputs/In/nState4 <-> WcState/WcState
//     Enc/Inputs/In/nState5 <-> Inputs/Touch probe status
//     Enc/Inputs/In/nState6 <-> Inputs/Touch probe status @bit 8
//     Enc/Outputs/Out/nCtrl5 <-> Outputs/Touch probe function
//     Enc/Outputs/Out/nCtrl6 <-> Outputs/Touch probe function @bit 8
//   NC-Task 1 SAF/Axes/Axis059_11 P2M1_CaCarryingWhirling1 <-> Device 3 (EtherCAT)/P2M1负极送片搬运1旋转 [11](InoSV660N)
//     Drive/Inputs/In/nDataIn1 <-> Inputs/Following error actual value
//     Drive/Inputs/In/nDcOutputTime <-> InfoData/DcOutputShift
//     Drive/Inputs/In/nState1 <-> Inputs/Statusword
//     Drive/Inputs/In/nState2 <-> Inputs/Statusword @bit 8
//     Drive/Inputs/In/nState4 @bit 1 <-> WcState/InputToggle
//     Drive/Inputs/In/nState4 <-> WcState/WcState
//     Drive/Outputs/Out/nCtrl1 <-> Outputs/Controlword
//     Drive/Outputs/Out/nCtrl2 <-> Outputs/Controlword @bit 8
//     Drive/Outputs/Out/nDataOut1 <-> Outputs/Target position
//     Enc/Inputs/In/nDataIn1 <-> Inputs/Position actual value
//     Enc/Inputs/In/nDataIn3 <-> Inputs/Touch probe pos1 pos value
//     Enc/Inputs/In/nDataIn5 <-> Inputs/Touch probe pos2 pos value
//     Enc/Inputs/In/nDcInputTime <-> InfoData/DcInputShift
//     Enc/Inputs/In/nState4 @bit 1 <-> WcState/InputToggle
//     Enc/Inputs/In/nState4 <-> WcState/WcState
//     Enc/Inputs/In/nState5 <-> Inputs/Touch probe status
//     Enc/Inputs/In/nState6 <-> Inputs/Touch probe status @bit 8
//     Enc/Outputs/Out/nCtrl5 <-> Outputs/Touch probe function
//     Enc/Outputs/Out/nCtrl6 <-> Outputs/Touch probe function @bit 8
//   NC-Task 1 SAF/Axes/Axis060_12 P2M1_CaCarryingLine2 <-> Device 3 (EtherCAT)/P2M1负极送片搬运2平移[12](CDHD)
//     Drive/Inputs/In/nDataIn1 <-> TxPDO 4/Following Error Actual Value
//     Drive/Inputs/In/nDcOutputTime <-> InfoData/DcOutputShift
//     Drive/Inputs/In/nState1 <-> TxPDO 1/StatusWord
//     Drive/Inputs/In/nState2 <-> TxPDO 1/StatusWord @bit 8
//     Drive/Inputs/In/nState4 @bit 1 <-> WcState/InputToggle
//     Drive/Inputs/In/nState4 <-> WcState/WcState
//     Drive/Inputs/In/nState5 <-> TxPDO 1/Modes of operation display
//     Drive/Outputs/Out/nCtrl1 <-> RxPDO 1/ControlWord
//     Drive/Outputs/Out/nCtrl2 <-> RxPDO 1/ControlWord @bit 8
//     Drive/Outputs/Out/nCtrl5 <-> RxPDO 1/Modes of operation
//     Drive/Outputs/Out/nDataOut1 <-> RxPDO 2/Target position
//     Drive/Outputs/Out/nDataOut2 <-> RxPDO 3/Target Velocity
//     Drive/Outputs/Out/nDataOut3[0] <-> RxPDO 4/Torque Offset
//     Drive/Outputs/Out/nDataOut4[0] <-> RxPDO 4/Target torque
//     Enc/Inputs/In/nDataIn1 <-> TxPDO 2/Position actual value
//     Enc/Inputs/In/nDcInputTime <-> InfoData/DcInputShift
//     Enc/Inputs/In/nState4 @bit 1 <-> WcState/InputToggle
//     Enc/Inputs/In/nState4 <-> WcState/WcState
//   NC-Task 1 SAF/Axes/Axis061_13 P2M1_CaCarryingUpDown2 <-> Device 3 (EtherCAT)/P2M1负极送片搬运2升降[13] (InoSV660N)
//     Drive/Inputs/In/nDataIn1 <-> Inputs/Following error actual value
//     Drive/Inputs/In/nDcOutputTime <-> InfoData/DcOutputShift
//     Drive/Inputs/In/nState1 <-> Inputs/Statusword
//     Drive/Inputs/In/nState2 <-> Inputs/Statusword @bit 8
//     Drive/Inputs/In/nState4 @bit 1 <-> WcState/InputToggle
//     Drive/Inputs/In/nState4 <-> WcState/WcState
//     Drive/Outputs/Out/nCtrl1 <-> Outputs/Controlword
//     Drive/Outputs/Out/nCtrl2 <-> Outputs/Controlword @bit 8
//     Drive/Outputs/Out/nDataOut1 <-> Outputs/Target position
//     Enc/Inputs/In/nDataIn1 <-> Inputs/Position actual value
//     Enc/Inputs/In/nDataIn3 <-> Inputs/Touch probe pos1 pos value
//     Enc/Inputs/In/nDataIn5 <-> Inputs/Touch probe pos2 pos value
//     Enc/Inputs/In/nDcInputTime <-> InfoData/DcInputShift
//     Enc/Inputs/In/nState4 @bit 1 <-> WcState/InputToggle
//     Enc/Inputs/In/nState4 <-> WcState/WcState
//     Enc/Inputs/In/nState5 <-> Inputs/Touch probe status
//     Enc/Inputs/In/nState6 <-> Inputs/Touch probe status @bit 8
//     Enc/Outputs/Out/nCtrl5 <-> Outputs/Touch probe function
//     Enc/Outputs/Out/nCtrl6 <-> Outputs/Touch probe function @bit 8
//   NC-Task 1 SAF/Axes/Axis062_14 P2M1_CaBelt <-> Device 3 (EtherCAT)/P2M1负极送片皮带[14](InoSV660N)
//     Drive/Inputs/In/nDataIn1 <-> Inputs/Following error actual value
//     Drive/Inputs/In/nDcOutputTime <-> InfoData/DcOutputShift
//     Drive/Inputs/In/nState1 <-> Inputs/Statusword
//     Drive/Inputs/In/nState2 <-> Inputs/Statusword @bit 8
//     Drive/Inputs/In/nState4 @bit 1 <-> WcState/InputToggle
//     Drive/Inputs/In/nState4 <-> WcState/WcState
//     Drive/Outputs/Out/nCtrl1 <-> Outputs/Controlword
//     Drive/Outputs/Out/nCtrl2 <-> Outputs/Controlword @bit 8
//     Drive/Outputs/Out/nDataOut1 <-> Outputs/Target position
//     Enc/Inputs/In/nDataIn1 <-> Inputs/Position actual value
//     Enc/Inputs/In/nDataIn3 <-> Inputs/Touch probe pos1 pos value
//     Enc/Inputs/In/nDataIn5 <-> Inputs/Touch probe pos2 pos value
//     Enc/Inputs/In/nDcInputTime <-> InfoData/DcInputShift
//     Enc/Inputs/In/nState4 @bit 1 <-> WcState/InputToggle
//     Enc/Inputs/In/nState4 <-> WcState/WcState
//     Enc/Inputs/In/nState5 <-> Inputs/Touch probe status
//     Enc/Inputs/In/nState6 <-> Inputs/Touch probe status @bit 8
//     Enc/Outputs/Out/nCtrl5 <-> Outputs/Touch probe function
//     Enc/Outputs/Out/nCtrl6 <-> Outputs/Touch probe function @bit 8
//   NC-Task 1 SAF/Axes/Axis063_15 P2M1_CaDTCarryingLine <-> Device 3 (EtherCAT)/P2M1负极叠台搬运平移[15](CDHD)
//     Drive/Inputs/In/nDataIn1 <-> TxPDO 4/Following Error Actual Value
//     Drive/Inputs/In/nDcOutputTime <-> InfoData/DcOutputShift
//     Drive/Inputs/In/nState1 <-> TxPDO 1/StatusWord
//     Drive/Inputs/In/nState2 <-> TxPDO 1/StatusWord @bit 8
//     Drive/Inputs/In/nState4 @bit 1 <-> WcState/InputToggle
//     Drive/Inputs/In/nState4 <-> WcState/WcState
//     Drive/Inputs/In/nState5 <-> TxPDO 1/Modes of operation display
//     Drive/Outputs/Out/nCtrl1 <-> RxPDO 1/ControlWord
//     Drive/Outputs/Out/nCtrl2 <-> RxPDO 1/ControlWord @bit 8
//     Drive/Outputs/Out/nCtrl5 <-> RxPDO 1/Modes of operation
//     Drive/Outputs/Out/nDataOut1 <-> RxPDO 2/Target position
//     Drive/Outputs/Out/nDataOut2 <-> RxPDO 3/Target Velocity
//     Drive/Outputs/Out/nDataOut3[0] <-> RxPDO 4/Torque Offset
//     Drive/Outputs/Out/nDataOut4[0] <-> RxPDO 4/Target torque
//     Enc/Inputs/In/nDataIn1 <-> TxPDO 2/Position actual value
//     Enc/Inputs/In/nDcInputTime <-> InfoData/DcInputShift
//     Enc/Inputs/In/nState4 @bit 1 <-> WcState/InputToggle
//     Enc/Inputs/In/nState4 <-> WcState/WcState
//   NC-Task 1 SAF/Axes/Axis064_16 P2M1_CaDTCarryingUpDown <-> Device 3 (EtherCAT)/P2M1负极叠台搬运升降[16](InoSV660N)
//     Drive/Inputs/In/nDataIn1 <-> Inputs/Following error actual value
//     Drive/Inputs/In/nDcOutputTime <-> InfoData/DcOutputShift
//     Drive/Inputs/In/nState1 <-> Inputs/Statusword
//     Drive/Inputs/In/nState2 <-> Inputs/Statusword @bit 8
//     Drive/Inputs/In/nState4 @bit 1 <-> WcState/InputToggle
//     Drive/Inputs/In/nState4 <-> WcState/WcState
//     Drive/Outputs/Out/nCtrl1 <-> Outputs/Controlword
//     Drive/Outputs/Out/nCtrl2 <-> Outputs/Controlword @bit 8
//     Drive/Outputs/Out/nDataOut1 <-> Outputs/Target position
//     Enc/Inputs/In/nDataIn1 <-> Inputs/Position actual value
//     Enc/Inputs/In/nDataIn3 <-> Inputs/Touch probe pos1 pos value
//     Enc/Inputs/In/nDataIn5 <-> Inputs/Touch probe pos2 pos value
//     Enc/Inputs/In/nDcInputTime <-> InfoData/DcInputShift
//     Enc/Inputs/In/nState4 @bit 1 <-> WcState/InputToggle
//     Enc/Inputs/In/nState4 <-> WcState/WcState
//     Enc/Inputs/In/nState5 <-> Inputs/Touch probe status
//     Enc/Inputs/In/nState6 <-> Inputs/Touch probe status @bit 8
//     Enc/Outputs/Out/nCtrl5 <-> Outputs/Touch probe function
//     Enc/Outputs/Out/nCtrl6 <-> Outputs/Touch probe function @bit 8
//   NC-Task 1 SAF/Axes/Axis065_17 P2M1_CadeviationX1 <-> Device 3 (EtherCAT)/P2M1负极纠偏平台X1[17] (InoSV660N)
//     Drive/Inputs/In/nDataIn1 <-> Inputs/Following error actual value
//     Drive/Inputs/In/nDcOutputTime <-> InfoData/DcOutputShift
//     Drive/Inputs/In/nState1 <-> Inputs/Statusword
//     Drive/Inputs/In/nState2 <-> Inputs/Statusword @bit 8
//     Drive/Inputs/In/nState4 @bit 1 <-> WcState/InputToggle
//     Drive/Inputs/In/nState4 <-> WcState/WcState
//     Drive/Outputs/Out/nCtrl1 <-> Outputs/Controlword
//     Drive/Outputs/Out/nCtrl2 <-> Outputs/Controlword @bit 8
//     Drive/Outputs/Out/nDataOut1 <-> Outputs/Target position
//     Enc/Inputs/In/nDataIn1 <-> Inputs/Position actual value
//     Enc/Inputs/In/nDataIn3 <-> Inputs/Touch probe pos1 pos value
//     Enc/Inputs/In/nDataIn5 <-> Inputs/Touch probe pos2 pos value
//     Enc/Inputs/In/nDcInputTime <-> InfoData/DcInputShift
//     Enc/Inputs/In/nState4 @bit 1 <-> WcState/InputToggle
//     Enc/Inputs/In/nState4 <-> WcState/WcState
//     Enc/Inputs/In/nState5 <-> Inputs/Touch probe status
//     Enc/Inputs/In/nState6 <-> Inputs/Touch probe status @bit 8
//     Enc/Outputs/Out/nCtrl5 <-> Outputs/Touch probe function
//     Enc/Outputs/Out/nCtrl6 <-> Outputs/Touch probe function @bit 8
//   NC-Task 1 SAF/Axes/Axis066_18 P2M1_CadeviationX2 <-> Device 3 (EtherCAT)/P2M1负极纠偏平台X2[18] (InoSV660N)
//     Drive/Inputs/In/nDataIn1 <-> Inputs/Following error actual value
//     Drive/Inputs/In/nDcOutputTime <-> InfoData/DcOutputShift
//     Drive/Inputs/In/nState1 <-> Inputs/Statusword
//     Drive/Inputs/In/nState2 <-> Inputs/Statusword @bit 8
//     Drive/Inputs/In/nState4 @bit 1 <-> WcState/InputToggle
//     Drive/Inputs/In/nState4 <-> WcState/WcState
//     Drive/Outputs/Out/nCtrl1 <-> Outputs/Controlword
//     Drive/Outputs/Out/nCtrl2 <-> Outputs/Controlword @bit 8
//     Drive/Outputs/Out/nDataOut1 <-> Outputs/Target position
//     Enc/Inputs/In/nDataIn1 <-> Inputs/Position actual value
//     Enc/Inputs/In/nDataIn3 <-> Inputs/Touch probe pos1 pos value
//     Enc/Inputs/In/nDataIn5 <-> Inputs/Touch probe pos2 pos value
//     Enc/Inputs/In/nDcInputTime <-> InfoData/DcInputShift
//     Enc/Inputs/In/nState4 @bit 1 <-> WcState/InputToggle
//     Enc/Inputs/In/nState4 <-> WcState/WcState
//     Enc/Inputs/In/nState5 <-> Inputs/Touch probe status
//     Enc/Inputs/In/nState6 <-> Inputs/Touch probe status @bit 8
//     Enc/Outputs/Out/nCtrl5 <-> Outputs/Touch probe function
//     Enc/Outputs/Out/nCtrl6 <-> Outputs/Touch probe function @bit 8
//   NC-Task 1 SAF/Axes/Axis067_19 P2M1_CadeviationY <-> Device 3 (EtherCAT)/P2M1负极纠偏平台Y [19](InoSV660N)
//     Drive/Inputs/In/nDataIn1 <-> Inputs/Following error actual value
//     Drive/Inputs/In/nDcOutputTime <-> InfoData/DcOutputShift
//     Drive/Inputs/In/nState1 <-> Inputs/Statusword
//     Drive/Inputs/In/nState2 <-> Inputs/Statusword @bit 8
//     Drive/Inputs/In/nState4 @bit 1 <-> WcState/InputToggle
//     Drive/Inputs/In/nState4 <-> WcState/WcState
//     Drive/Outputs/Out/nCtrl1 <-> Outputs/Controlword
//     Drive/Outputs/Out/nCtrl2 <-> Outputs/Controlword @bit 8
//     Drive/Outputs/Out/nDataOut1 <-> Outputs/Target position
//     Enc/Inputs/In/nDataIn1 <-> Inputs/Position actual value
//     Enc/Inputs/In/nDataIn3 <-> Inputs/Touch probe pos1 pos value
//     Enc/Inputs/In/nDataIn5 <-> Inputs/Touch probe pos2 pos value
//     Enc/Inputs/In/nDcInputTime <-> InfoData/DcInputShift
//     Enc/Inputs/In/nState4 @bit 1 <-> WcState/InputToggle
//     Enc/Inputs/In/nState4 <-> WcState/WcState
//     Enc/Inputs/In/nState5 <-> Inputs/Touch probe status
//     Enc/Inputs/In/nState6 <-> Inputs/Touch probe status @bit 8
//     Enc/Outputs/Out/nCtrl5 <-> Outputs/Touch probe function
//     Enc/Outputs/Out/nCtrl6 <-> Outputs/Touch probe function @bit 8
//   NC-Task 1 SAF/Axes/Axis068_20 P2M1_SEPTAunwinding <-> Device 3 (EtherCAT)/P2M1隔膜放卷[20] (InoSV660N)
//     Drive/Inputs/In/nDataIn1 <-> Inputs/Following error actual value
//     Drive/Inputs/In/nDcOutputTime <-> InfoData/DcOutputShift
//     Drive/Inputs/In/nState1 <-> Inputs/Statusword
//     Drive/Inputs/In/nState2 <-> Inputs/Statusword @bit 8
//     Drive/Inputs/In/nState4 @bit 1 <-> WcState/InputToggle
//     Drive/Inputs/In/nState4 <-> WcState/WcState
//     Drive/Outputs/Out/nCtrl1 <-> Outputs/Controlword
//     Drive/Outputs/Out/nCtrl2 <-> Outputs/Controlword @bit 8
//     Drive/Outputs/Out/nDataOut1 <-> Outputs/Target position
//     Enc/Inputs/In/nDataIn1 <-> Inputs/Position actual value
//     Enc/Inputs/In/nDataIn3 <-> Inputs/Touch probe pos1 pos value
//     Enc/Inputs/In/nDataIn5 <-> Inputs/Touch probe pos2 pos value
//     Enc/Inputs/In/nDcInputTime <-> InfoData/DcInputShift
//     Enc/Inputs/In/nState4 @bit 1 <-> WcState/InputToggle
//     Enc/Inputs/In/nState4 <-> WcState/WcState
//     Enc/Inputs/In/nState5 <-> Inputs/Touch probe status
//     Enc/Inputs/In/nState6 <-> Inputs/Touch probe status @bit 8
//     Enc/Outputs/Out/nCtrl5 <-> Outputs/Touch probe function
//     Enc/Outputs/Out/nCtrl6 <-> Outputs/Touch probe function @bit 8
//   NC-Task 1 SAF/Axes/Axis069_21 P2M1_SEPTAdeviation1 <-> Device 3 (EtherCAT)/P2M1隔膜放卷纠偏_[21](InoSV660N)
//     Drive/Inputs/In/nDataIn1 <-> Inputs/Following error actual value
//     Drive/Inputs/In/nDcOutputTime <-> InfoData/DcOutputShift
//     Drive/Inputs/In/nState1 <-> Inputs/Statusword
//     Drive/Inputs/In/nState2 <-> Inputs/Statusword @bit 8
//     Drive/Inputs/In/nState4 @bit 1 <-> WcState/InputToggle
//     Drive/Inputs/In/nState4 <-> WcState/WcState
//     Drive/Outputs/Out/nCtrl1 <-> Outputs/Controlword
//     Drive/Outputs/Out/nCtrl2 <-> Outputs/Controlword @bit 8
//     Drive/Outputs/Out/nDataOut1 <-> Outputs/Target position
//     Enc/Inputs/In/nDataIn1 <-> Inputs/Position actual value
//     Enc/Inputs/In/nDataIn3 <-> Inputs/Touch probe pos1 pos value
//     Enc/Inputs/In/nDataIn5 <-> Inputs/Touch probe pos2 pos value
//     Enc/Inputs/In/nDcInputTime <-> InfoData/DcInputShift
//     Enc/Inputs/In/nState4 @bit 1 <-> WcState/InputToggle
//     Enc/Inputs/In/nState4 <-> WcState/WcState
//     Enc/Inputs/In/nState5 <-> Inputs/Touch probe status
//     Enc/Inputs/In/nState6 <-> Inputs/Touch probe status @bit 8
//     Enc/Outputs/Out/nCtrl5 <-> Outputs/Touch probe function
//     Enc/Outputs/Out/nCtrl6 <-> Outputs/Touch probe function @bit 8
//   NC-Task 1 SAF/Axes/Axis070_22 P2M1_SEPTAdeviation2 <-> Device 3 (EtherCAT)/P2M1隔膜尾部纠偏[22] (InoSV660N)
//     Drive/Inputs/In/nDataIn1 <-> Inputs/Following error actual value
//     Drive/Inputs/In/nDcOutputTime <-> InfoData/DcOutputShift
//     Drive/Inputs/In/nState1 <-> Inputs/Statusword
//     Drive/Inputs/In/nState2 <-> Inputs/Statusword @bit 8
//     Drive/Inputs/In/nState4 @bit 1 <-> WcState/InputToggle
//     Drive/Inputs/In/nState4 <-> WcState/WcState
//     Drive/Outputs/Out/nCtrl1 <-> Outputs/Controlword
//     Drive/Outputs/Out/nCtrl2 <-> Outputs/Controlword @bit 8
//     Drive/Outputs/Out/nDataOut1 <-> Outputs/Target position
//     Enc/Inputs/In/nDataIn1 <-> Inputs/Position actual value
//     Enc/Inputs/In/nDataIn3 <-> Inputs/Touch probe pos1 pos value
//     Enc/Inputs/In/nDataIn5 <-> Inputs/Touch probe pos2 pos value
//     Enc/Inputs/In/nDcInputTime <-> InfoData/DcInputShift
//     Enc/Inputs/In/nState4 @bit 1 <-> WcState/InputToggle
//     Enc/Inputs/In/nState4 <-> WcState/WcState
//     Enc/Inputs/In/nState5 <-> Inputs/Touch probe status
//     Enc/Inputs/In/nState6 <-> Inputs/Touch probe status @bit 8
//     Enc/Outputs/Out/nCtrl5 <-> Outputs/Touch probe function
//     Enc/Outputs/Out/nCtrl6 <-> Outputs/Touch probe function @bit 8
//   NC-Task 1 SAF/Axes/Axis071_23 P2M1_SEPTATension <-> Device 3 (EtherCAT)/P2M1隔膜摆杆张力[23] (InoSV660N)
//     Drive/Inputs/In/nDcOutputTime <-> InfoData/DcOutputShift
//     Drive/Inputs/In/nState1 <-> Inputs/Statusword
//     Drive/Inputs/In/nState2 <-> Inputs/Statusword @bit 8
//     Drive/Inputs/In/nState4 @bit 1 <-> WcState/InputToggle
//     Drive/Inputs/In/nState4 <-> WcState/WcState
//     Drive/Inputs/In/nState5 <-> Inputs/Modes of operation display
//     Drive/Outputs/Out/nCtrl1 <-> Outputs/Controlword
//     Drive/Outputs/Out/nCtrl2 <-> Outputs/Controlword @bit 8
//     Drive/Outputs/Out/nDataOut1 <-> Outputs/Target position
//     Drive/Outputs/Out/nDataOut2 <-> Outputs/Target velocity
//     Enc/Inputs/In/nDataIn1 <-> Inputs/Position actual value
//     Enc/Inputs/In/nDataIn3 <-> Inputs/Touch probe pos1 pos value
//     Enc/Inputs/In/nDataIn5 <-> Inputs/Touch probe pos2 pos value
//     Enc/Inputs/In/nDcInputTime <-> InfoData/DcInputShift
//     Enc/Inputs/In/nState4 @bit 1 <-> WcState/InputToggle
//     Enc/Inputs/In/nState4 <-> WcState/WcState
//     Enc/Inputs/In/nState5 <-> Inputs/Touch probe status
//     Enc/Inputs/In/nState6 <-> Inputs/Touch probe status @bit 8
//     Enc/Outputs/Out/nCtrl5 <-> Outputs/Touch probe function
//     Enc/Outputs/Out/nCtrl6 <-> Outputs/Touch probe function @bit 8
//   NC-Task 1 SAF/Axes/Axis072_24 P2M1_SEPTATCache <-> Device 3 (EtherCAT)/P2M1隔膜缓存[24](CDHD)
//     Drive/Inputs/In/nDataIn1 <-> TxPDO 4/Following Error Actual Value
//     Drive/Inputs/In/nDcOutputTime <-> InfoData/DcOutputShift
//     Drive/Inputs/In/nState1 <-> TxPDO 1/StatusWord
//     Drive/Inputs/In/nState2 <-> TxPDO 1/StatusWord @bit 8
//     Drive/Inputs/In/nState4 @bit 1 <-> WcState/InputToggle
//     Drive/Inputs/In/nState4 <-> WcState/WcState
//     Drive/Inputs/In/nState5 <-> TxPDO 1/Modes of operation display
//     Drive/Outputs/Out/nCtrl1 <-> RxPDO 1/ControlWord
//     Drive/Outputs/Out/nCtrl2 <-> RxPDO 1/ControlWord @bit 8
//     Drive/Outputs/Out/nCtrl5 <-> RxPDO 1/Modes of operation
//     Drive/Outputs/Out/nDataOut1 <-> RxPDO 2/Target position
//     Drive/Outputs/Out/nDataOut2 <-> RxPDO 3/Target Velocity
//     Drive/Outputs/Out/nDataOut3[0] <-> RxPDO 4/Torque Offset
//     Drive/Outputs/Out/nDataOut4[0] <-> RxPDO 4/Target torque
//     Enc/Inputs/In/nDataIn1 <-> TxPDO 2/Position actual value
//     Enc/Inputs/In/nDcInputTime <-> InfoData/DcInputShift
//     Enc/Inputs/In/nState4 @bit 1 <-> WcState/InputToggle
//     Enc/Inputs/In/nState4 <-> WcState/WcState
//   NC-Task 1 SAF/Axes/Axis073_25 P2M1_SEPTATLine <-> Device 3 (EtherCAT)/P2M1隔膜平移[25](CDHD)
//     Drive/Inputs/In/nDataIn1 <-> TxPDO 4/Following Error Actual Value
//     Drive/Inputs/In/nDcOutputTime <-> InfoData/DcOutputShift
//     Drive/Inputs/In/nState1 <-> TxPDO 1/StatusWord
//     Drive/Inputs/In/nState2 <-> TxPDO 1/StatusWord @bit 8
//     Drive/Inputs/In/nState4 @bit 1 <-> WcState/InputToggle
//     Drive/Inputs/In/nState4 <-> WcState/WcState
//     Drive/Inputs/In/nState5 <-> TxPDO 1/Modes of operation display
//     Drive/Outputs/Out/nCtrl1 <-> RxPDO 1/ControlWord
//     Drive/Outputs/Out/nCtrl2 <-> RxPDO 1/ControlWord @bit 8
//     Drive/Outputs/Out/nCtrl5 <-> RxPDO 1/Modes of operation
//     Drive/Outputs/Out/nDataOut1 <-> RxPDO 2/Target position
//     Drive/Outputs/Out/nDataOut2 <-> RxPDO 3/Target Velocity
//     Drive/Outputs/Out/nDataOut3[0] <-> RxPDO 4/Torque Offset
//     Drive/Outputs/Out/nDataOut4[0] <-> RxPDO 4/Target torque
//     Enc/Inputs/In/nDataIn1 <-> TxPDO 2/Position actual value
//     Enc/Inputs/In/nDcInputTime <-> InfoData/DcInputShift
//     Enc/Inputs/In/nState4 @bit 1 <-> WcState/InputToggle
//     Enc/Inputs/In/nState4 <-> WcState/WcState
//   NC-Task 1 SAF/Axes/Axis074_26 P2M1_DTUpDown <-> Device 3 (EtherCAT)/P2M1叠台升降[26] (InoSV660N)
//     Drive/Inputs/In/nDataIn1 <-> Inputs/Following error actual value
//     Drive/Inputs/In/nDcOutputTime <-> InfoData/DcOutputShift
//     Drive/Inputs/In/nState1 <-> Inputs/Statusword
//     Drive/Inputs/In/nState2 <-> Inputs/Statusword @bit 8
//     Drive/Inputs/In/nState4 @bit 1 <-> WcState/InputToggle
//     Drive/Inputs/In/nState4 <-> WcState/WcState
//     Drive/Outputs/Out/nCtrl1 <-> Outputs/Controlword
//     Drive/Outputs/Out/nCtrl2 <-> Outputs/Controlword @bit 8
//     Drive/Outputs/Out/nDataOut1 <-> Outputs/Target position
//     Enc/Inputs/In/nDataIn1 <-> Inputs/Position actual value
//     Enc/Inputs/In/nDataIn3 <-> Inputs/Touch probe pos1 pos value
//     Enc/Inputs/In/nDataIn5 <-> Inputs/Touch probe pos2 pos value
//     Enc/Inputs/In/nDcInputTime <-> InfoData/DcInputShift
//     Enc/Inputs/In/nState4 @bit 1 <-> WcState/InputToggle
//     Enc/Inputs/In/nState4 <-> WcState/WcState
//     Enc/Inputs/In/nState5 <-> Inputs/Touch probe status
//     Enc/Inputs/In/nState6 <-> Inputs/Touch probe status @bit 8
//     Enc/Outputs/Out/nCtrl5 <-> Outputs/Touch probe function
//     Enc/Outputs/Out/nCtrl6 <-> Outputs/Touch probe function @bit 8
//   NC-Task 1 SAF/Axes/Axis075_27 P2M1_LeftYDLine <-> Device 3 (EtherCAT)/P2M1左压刀开合[27] (InoSV660N)
//     Drive/Inputs/In/nDataIn1 <-> Inputs/Following error actual value
//     Drive/Inputs/In/nDcOutputTime <-> InfoData/DcOutputShift
//     Drive/Inputs/In/nState1 <-> Inputs/Statusword
//     Drive/Inputs/In/nState2 <-> Inputs/Statusword @bit 8
//     Drive/Inputs/In/nState4 @bit 1 <-> WcState/InputToggle
//     Drive/Inputs/In/nState4 <-> WcState/WcState
//     Drive/Outputs/Out/nCtrl1 <-> Outputs/Controlword
//     Drive/Outputs/Out/nCtrl2 <-> Outputs/Controlword @bit 8
//     Drive/Outputs/Out/nDataOut1 <-> Outputs/Target position
//     Enc/Inputs/In/nDataIn1 <-> Inputs/Position actual value
//     Enc/Inputs/In/nDataIn3 <-> Inputs/Touch probe pos1 pos value
//     Enc/Inputs/In/nDataIn5 <-> Inputs/Touch probe pos2 pos value
//     Enc/Inputs/In/nDcInputTime <-> InfoData/DcInputShift
//     Enc/Inputs/In/nState4 @bit 1 <-> WcState/InputToggle
//     Enc/Inputs/In/nState4 <-> WcState/WcState
//     Enc/Inputs/In/nState5 <-> Inputs/Touch probe status
//     Enc/Inputs/In/nState6 <-> Inputs/Touch probe status @bit 8
//     Enc/Outputs/Out/nCtrl5 <-> Outputs/Touch probe function
//     Enc/Outputs/Out/nCtrl6 <-> Outputs/Touch probe function @bit 8
//   NC-Task 1 SAF/Axes/Axis076_28 P2M1_LeftYDUpDown <-> Device 3 (EtherCAT)/P2M1左压刀升降[28] (InoSV660N)
//     Drive/Inputs/In/nDataIn1 <-> Inputs/Following error actual value
//     Drive/Inputs/In/nDcOutputTime <-> InfoData/DcOutputShift
//     Drive/Inputs/In/nState1 <-> Inputs/Statusword
//     Drive/Inputs/In/nState2 <-> Inputs/Statusword @bit 8
//     Drive/Inputs/In/nState4 @bit 1 <-> WcState/InputToggle
//     Drive/Inputs/In/nState4 <-> WcState/WcState
//     Drive/Outputs/Out/nCtrl1 <-> Outputs/Controlword
//     Drive/Outputs/Out/nCtrl2 <-> Outputs/Controlword @bit 8
//     Drive/Outputs/Out/nDataOut1 <-> Outputs/Target position
//     Enc/Inputs/In/nDataIn1 <-> Inputs/Position actual value
//     Enc/Inputs/In/nDataIn3 <-> Inputs/Touch probe pos1 pos value
//     Enc/Inputs/In/nDataIn5 <-> Inputs/Touch probe pos2 pos value
//     Enc/Inputs/In/nDcInputTime <-> InfoData/DcInputShift
//     Enc/Inputs/In/nState4 @bit 1 <-> WcState/InputToggle
//     Enc/Inputs/In/nState4 <-> WcState/WcState
//     Enc/Inputs/In/nState5 <-> Inputs/Touch probe status
//     Enc/Inputs/In/nState6 <-> Inputs/Touch probe status @bit 8
//     Enc/Outputs/Out/nCtrl5 <-> Outputs/Touch probe function
//     Enc/Outputs/Out/nCtrl6 <-> Outputs/Touch probe function @bit 8
//   NC-Task 1 SAF/Axes/Axis077_29 P2M1_RightYDLine <-> Device 3 (EtherCAT)/P2M1右压刀开合 [29](InoSV660N)
//     Drive/Inputs/In/nDataIn1 <-> Inputs/Following error actual value
//     Drive/Inputs/In/nDcOutputTime <-> InfoData/DcOutputShift
//     Drive/Inputs/In/nState1 <-> Inputs/Statusword
//     Drive/Inputs/In/nState2 <-> Inputs/Statusword @bit 8
//     Drive/Inputs/In/nState4 @bit 1 <-> WcState/InputToggle
//     Drive/Inputs/In/nState4 <-> WcState/WcState
//     Drive/Outputs/Out/nCtrl1 <-> Outputs/Controlword
//     Drive/Outputs/Out/nCtrl2 <-> Outputs/Controlword @bit 8
//     Drive/Outputs/Out/nDataOut1 <-> Outputs/Target position
//     Enc/Inputs/In/nDataIn1 <-> Inputs/Position actual value
//     Enc/Inputs/In/nDataIn3 <-> Inputs/Touch probe pos1 pos value
//     Enc/Inputs/In/nDataIn5 <-> Inputs/Touch probe pos2 pos value
//     Enc/Inputs/In/nDcInputTime <-> InfoData/DcInputShift
//     Enc/Inputs/In/nState4 @bit 1 <-> WcState/InputToggle
//     Enc/Inputs/In/nState4 <-> WcState/WcState
//     Enc/Inputs/In/nState5 <-> Inputs/Touch probe status
//     Enc/Inputs/In/nState6 <-> Inputs/Touch probe status @bit 8
//     Enc/Outputs/Out/nCtrl5 <-> Outputs/Touch probe function
//     Enc/Outputs/Out/nCtrl6 <-> Outputs/Touch probe function @bit 8
//   NC-Task 1 SAF/Axes/Axis078_30 P2M1_RightYDUpDown <-> Device 3 (EtherCAT)/P2M1右压刀升降[30] (InoSV660N)
//     Drive/Inputs/In/nDataIn1 <-> Inputs/Following error actual value
//     Drive/Inputs/In/nDcOutputTime <-> InfoData/DcOutputShift
//     Drive/Inputs/In/nState1 <-> Inputs/Statusword
//     Drive/Inputs/In/nState2 <-> Inputs/Statusword @bit 8
//     Drive/Inputs/In/nState4 @bit 1 <-> WcState/InputToggle
//     Drive/Inputs/In/nState4 <-> WcState/WcState
//     Drive/Outputs/Out/nCtrl1 <-> Outputs/Controlword
//     Drive/Outputs/Out/nCtrl2 <-> Outputs/Controlword @bit 8
//     Drive/Outputs/Out/nDataOut1 <-> Outputs/Target position
//     Enc/Inputs/In/nDataIn1 <-> Inputs/Position actual value
//     Enc/Inputs/In/nDataIn3 <-> Inputs/Touch probe pos1 pos value
//     Enc/Inputs/In/nDataIn5 <-> Inputs/Touch probe pos2 pos value
//     Enc/Inputs/In/nDcInputTime <-> InfoData/DcInputShift
//     Enc/Inputs/In/nState4 @bit 1 <-> WcState/InputToggle
//     Enc/Inputs/In/nState4 <-> WcState/WcState
//     Enc/Inputs/In/nState5 <-> Inputs/Touch probe status
//     Enc/Inputs/In/nState6 <-> Inputs/Touch probe status @bit 8
//     Enc/Outputs/Out/nCtrl5 <-> Outputs/Touch probe function
//     Enc/Outputs/Out/nCtrl6 <-> Outputs/Touch probe function @bit 8
//   NC-Task 1 SAF/Axes/Axis079_31 P2M1_TailCurlLine <-> Device 3 (EtherCAT)/P2M1尾卷夹电芯平移[31](InoSV660N)
//     Drive/Inputs/In/nDataIn1 <-> Inputs/Following error actual value
//     Drive/Inputs/In/nDcOutputTime <-> InfoData/DcOutputShift
//     Drive/Inputs/In/nState1 <-> Inputs/Statusword
//     Drive/Inputs/In/nState2 <-> Inputs/Statusword @bit 8
//     Drive/Inputs/In/nState4 @bit 1 <-> WcState/InputToggle
//     Drive/Inputs/In/nState4 <-> WcState/WcState
//     Drive/Outputs/Out/nCtrl1 <-> Outputs/Controlword
//     Drive/Outputs/Out/nCtrl2 <-> Outputs/Controlword @bit 8
//     Drive/Outputs/Out/nDataOut1 <-> Outputs/Target position
//     Enc/Inputs/In/nDataIn1 <-> Inputs/Position actual value
//     Enc/Inputs/In/nDataIn3 <-> Inputs/Touch probe pos1 pos value
//     Enc/Inputs/In/nDataIn5 <-> Inputs/Touch probe pos2 pos value
//     Enc/Inputs/In/nDcInputTime <-> InfoData/DcInputShift
//     Enc/Inputs/In/nState4 @bit 1 <-> WcState/InputToggle
//     Enc/Inputs/In/nState4 <-> WcState/WcState
//     Enc/Inputs/In/nState5 <-> Inputs/Touch probe status
//     Enc/Inputs/In/nState6 <-> Inputs/Touch probe status @bit 8
//     Enc/Outputs/Out/nCtrl5 <-> Outputs/Touch probe function
//     Enc/Outputs/Out/nCtrl6 <-> Outputs/Touch probe function @bit 8
//   NC-Task 1 SAF/Axes/Axis080_32 P2M1_TailCurlUpDown <-> Device 3 (EtherCAT)/P2M1尾卷夹电芯升降[32](InoSV660N)
//     Drive/Inputs/In/nDataIn1 <-> Inputs/Following error actual value
//     Drive/Inputs/In/nDcOutputTime <-> InfoData/DcOutputShift
//     Drive/Inputs/In/nState1 <-> Inputs/Statusword
//     Drive/Inputs/In/nState2 <-> Inputs/Statusword @bit 8
//     Drive/Inputs/In/nState4 @bit 1 <-> WcState/InputToggle
//     Drive/Inputs/In/nState4 <-> WcState/WcState
//     Drive/Outputs/Out/nCtrl1 <-> Outputs/Controlword
//     Drive/Outputs/Out/nCtrl2 <-> Outputs/Controlword @bit 8
//     Drive/Outputs/Out/nDataOut1 <-> Outputs/Target position
//     Enc/Inputs/In/nDataIn1 <-> Inputs/Position actual value
//     Enc/Inputs/In/nDataIn3 <-> Inputs/Touch probe pos1 pos value
//     Enc/Inputs/In/nDataIn5 <-> Inputs/Touch probe pos2 pos value
//     Enc/Inputs/In/nDcInputTime <-> InfoData/DcInputShift
//     Enc/Inputs/In/nState4 @bit 1 <-> WcState/InputToggle
//     Enc/Inputs/In/nState4 <-> WcState/WcState
//     Enc/Inputs/In/nState5 <-> Inputs/Touch probe status
//     Enc/Inputs/In/nState6 <-> Inputs/Touch probe status @bit 8
//     Enc/Outputs/Out/nCtrl5 <-> Outputs/Touch probe function
//     Enc/Outputs/Out/nCtrl6 <-> Outputs/Touch probe function @bit 8
//   NC-Task 1 SAF/Axes/Axis081_33 P2M1_TailCurlRetracting <-> Device 3 (EtherCAT)/P2M1尾卷夹电芯伸缩[33] (InoSV660N)
//     Drive/Inputs/In/nDataIn1 <-> Inputs/Following error actual value
//     Drive/Inputs/In/nDcOutputTime <-> InfoData/DcOutputShift
//     Drive/Inputs/In/nState1 <-> Inputs/Statusword
//     Drive/Inputs/In/nState2 <-> Inputs/Statusword @bit 8
//     Drive/Inputs/In/nState4 @bit 1 <-> WcState/InputToggle
//     Drive/Inputs/In/nState4 <-> WcState/WcState
//     Drive/Outputs/Out/nCtrl1 <-> Outputs/Controlword
//     Drive/Outputs/Out/nCtrl2 <-> Outputs/Controlword @bit 8
//     Drive/Outputs/Out/nDataOut1 <-> Outputs/Target position
//     Enc/Inputs/In/nDataIn1 <-> Inputs/Position actual value
//     Enc/Inputs/In/nDataIn3 <-> Inputs/Touch probe pos1 pos value
//     Enc/Inputs/In/nDataIn5 <-> Inputs/Touch probe pos2 pos value
//     Enc/Inputs/In/nDcInputTime <-> InfoData/DcInputShift
//     Enc/Inputs/In/nState4 @bit 1 <-> WcState/InputToggle
//     Enc/Inputs/In/nState4 <-> WcState/WcState
//     Enc/Inputs/In/nState5 <-> Inputs/Touch probe status
//     Enc/Inputs/In/nState6 <-> Inputs/Touch probe status @bit 8
//     Enc/Outputs/Out/nCtrl5 <-> Outputs/Touch probe function
//     Enc/Outputs/Out/nCtrl6 <-> Outputs/Touch probe function @bit 8
//   NC-Task 1 SAF/Axes/Axis082_34 P2M1_TailCurlWhirling <-> Device 3 (EtherCAT)/P2M1尾卷夹电芯旋转[34] (InoSV660N)
//     Drive/Inputs/In/nDataIn1 <-> Inputs/Following error actual value
//     Drive/Inputs/In/nDcOutputTime <-> InfoData/DcOutputShift
//     Drive/Inputs/In/nState1 <-> Inputs/Statusword
//     Drive/Inputs/In/nState2 <-> Inputs/Statusword @bit 8
//     Drive/Inputs/In/nState4 @bit 1 <-> WcState/InputToggle
//     Drive/Inputs/In/nState4 <-> WcState/WcState
//     Drive/Outputs/Out/nCtrl1 <-> Outputs/Controlword
//     Drive/Outputs/Out/nCtrl2 <-> Outputs/Controlword @bit 8
//     Drive/Outputs/Out/nDataOut1 <-> Outputs/Target position
//     Enc/Inputs/In/nDataIn1 <-> Inputs/Position actual value
//     Enc/Inputs/In/nDataIn3 <-> Inputs/Touch probe pos1 pos value
//     Enc/Inputs/In/nDataIn5 <-> Inputs/Touch probe pos2 pos value
//     Enc/Inputs/In/nDcInputTime <-> InfoData/DcInputShift
//     Enc/Inputs/In/nState4 @bit 1 <-> WcState/InputToggle
//     Enc/Inputs/In/nState4 <-> WcState/WcState
//     Enc/Inputs/In/nState5 <-> Inputs/Touch probe status
//     Enc/Inputs/In/nState6 <-> Inputs/Touch probe status @bit 8
//     Enc/Outputs/Out/nCtrl5 <-> Outputs/Touch probe function
//     Enc/Outputs/Out/nCtrl6 <-> Outputs/Touch probe function @bit 8
//   NC-Task 1 SAF/Axes/Axis083_35 P2M1_TailCurlSEPTALine <-> Device 3 (EtherCAT)/P2M1夹膜平移[35](InoSV660N)
//     Drive/Inputs/In/nDataIn1 <-> Inputs/Following error actual value
//     Drive/Inputs/In/nDcOutputTime <-> InfoData/DcOutputShift
//     Drive/Inputs/In/nState1 <-> Inputs/Statusword
//     Drive/Inputs/In/nState2 <-> Inputs/Statusword @bit 8
//     Drive/Inputs/In/nState4 @bit 1 <-> WcState/InputToggle
//     Drive/Inputs/In/nState4 <-> WcState/WcState
//     Drive/Outputs/Out/nCtrl1 <-> Outputs/Controlword
//     Drive/Outputs/Out/nCtrl2 <-> Outputs/Controlword @bit 8
//     Drive/Outputs/Out/nDataOut1 <-> Outputs/Target position
//     Enc/Inputs/In/nDataIn1 <-> Inputs/Position actual value
//     Enc/Inputs/In/nDataIn3 <-> Inputs/Touch probe pos1 pos value
//     Enc/Inputs/In/nDataIn5 <-> Inputs/Touch probe pos2 pos value
//     Enc/Inputs/In/nDcInputTime <-> InfoData/DcInputShift
//     Enc/Inputs/In/nState4 @bit 1 <-> WcState/InputToggle
//     Enc/Inputs/In/nState4 <-> WcState/WcState
//     Enc/Inputs/In/nState5 <-> Inputs/Touch probe status
//     Enc/Inputs/In/nState6 <-> Inputs/Touch probe status @bit 8
//     Enc/Outputs/Out/nCtrl5 <-> Outputs/Touch probe function
//     Enc/Outputs/Out/nCtrl6 <-> Outputs/Touch probe function @bit 8
//   NC-Task 1 SAF/Axes/Axis084_36 P2M1_TailCurlSEPTAUpDown <-> Device 3 (EtherCAT)/P2M1夹膜升降[36] (InoSV660N)
//     Drive/Inputs/In/nDataIn1 <-> Inputs/Following error actual value
//     Drive/Inputs/In/nDcOutputTime <-> InfoData/DcOutputShift
//     Drive/Inputs/In/nState1 <-> Inputs/Statusword
//     Drive/Inputs/In/nState2 <-> Inputs/Statusword @bit 8
//     Drive/Inputs/In/nState4 @bit 1 <-> WcState/InputToggle
//     Drive/Inputs/In/nState4 <-> WcState/WcState
//     Drive/Outputs/Out/nCtrl1 <-> Outputs/Controlword
//     Drive/Outputs/Out/nCtrl2 <-> Outputs/Controlword @bit 8
//     Drive/Outputs/Out/nDataOut1 <-> Outputs/Target position
//     Enc/Inputs/In/nDataIn1 <-> Inputs/Position actual value
//     Enc/Inputs/In/nDataIn3 <-> Inputs/Touch probe pos1 pos value
//     Enc/Inputs/In/nDataIn5 <-> Inputs/Touch probe pos2 pos value
//     Enc/Inputs/In/nDcInputTime <-> InfoData/DcInputShift
//     Enc/Inputs/In/nState4 @bit 1 <-> WcState/InputToggle
//     Enc/Inputs/In/nState4 <-> WcState/WcState
//     Enc/Inputs/In/nState5 <-> Inputs/Touch probe status
//     Enc/Inputs/In/nState6 <-> Inputs/Touch probe status @bit 8
//     Enc/Outputs/Out/nCtrl5 <-> Outputs/Touch probe function
//     Enc/Outputs/Out/nCtrl6 <-> Outputs/Touch probe function @bit 8
//   NC-Task 1 SAF/Axes/Axis085_37 P2M1_LCurlingneedleLine <-> Device 3 (EtherCAT)/P2M1长卷针平移[37](CL3C-EC808AC)
//     Drive/Inputs/In/nDcOutputTime <-> InfoData/DcOutputShift
//     Drive/Inputs/In/nState1 <-> Transmit PDO 1/Status Word
//     Drive/Inputs/In/nState2 <-> Transmit PDO 1/Status Word @bit 8
//     Drive/Inputs/In/nState4 @bit 1 <-> WcState/InputToggle
//     Drive/Inputs/In/nState4 <-> WcState/WcState
//     Drive/Outputs/Out/nCtrl1 <-> Receive PDO 1/Control Word
//     Drive/Outputs/Out/nCtrl2 <-> Receive PDO 1/Control Word @bit 8
//     Drive/Outputs/Out/nDataOut1 <-> Receive PDO 1/Profile Target Position
//     Enc/Inputs/In/nDataIn1 <-> Transmit PDO 1/Position Actual Value
//     Enc/Inputs/In/nDataIn3 <-> Transmit PDO 1/Touch Probe 1 Positive Value
//     Enc/Inputs/In/nDcInputTime <-> InfoData/DcInputShift
//     Enc/Inputs/In/nState4 @bit 1 <-> WcState/InputToggle
//     Enc/Inputs/In/nState4 <-> WcState/WcState
//     Enc/Inputs/In/nState5 <-> Transmit PDO 1/Touch Probe Status
//     Enc/Inputs/In/nState6 <-> Transmit PDO 1/Touch Probe Status @bit 8
//     Enc/Outputs/Out/nCtrl5 <-> Receive PDO 1/Touch Probe Function
//     Enc/Outputs/Out/nCtrl6 <-> Receive PDO 1/Touch Probe Function @bit 8
//   NC-Task 1 SAF/Axes/Axis086_38 P2M1_SCurlingneedleLine <-> Device 3 (EtherCAT)/P2M1短卷针平移[38](CL3C-EC808AC)
//     Drive/Inputs/In/nDcOutputTime <-> InfoData/DcOutputShift
//     Drive/Inputs/In/nState1 <-> Transmit PDO 1/Status Word
//     Drive/Inputs/In/nState2 <-> Transmit PDO 1/Status Word @bit 8
//     Drive/Inputs/In/nState4 @bit 1 <-> WcState/InputToggle
//     Drive/Inputs/In/nState4 <-> WcState/WcState
//     Drive/Outputs/Out/nCtrl1 <-> Receive PDO 1/Control Word
//     Drive/Outputs/Out/nCtrl2 <-> Receive PDO 1/Control Word @bit 8
//     Drive/Outputs/Out/nDataOut1 <-> Receive PDO 1/Profile Target Position
//     Enc/Inputs/In/nDataIn1 <-> Transmit PDO 1/Position Actual Value
//     Enc/Inputs/In/nDataIn3 <-> Transmit PDO 1/Touch Probe 1 Positive Value
//     Enc/Inputs/In/nDcInputTime <-> InfoData/DcInputShift
//     Enc/Inputs/In/nState4 @bit 1 <-> WcState/InputToggle
//     Enc/Inputs/In/nState4 <-> WcState/WcState
//     Enc/Inputs/In/nState5 <-> Transmit PDO 1/Touch Probe Status
//     Enc/Inputs/In/nState6 <-> Transmit PDO 1/Touch Probe Status @bit 8
//     Enc/Outputs/Out/nCtrl5 <-> Receive PDO 1/Touch Probe Function
//     Enc/Outputs/Out/nCtrl6 <-> Receive PDO 1/Touch Probe Function @bit 8
//   NC-Task 1 SAF/Axes/Axis087_39 P2M1_LCurlingneedleWhirling <-> Device 3 (EtherCAT)/P2M1长卷针旋转[39](CL3C-EC808AC)
//     Drive/Inputs/In/nDcOutputTime <-> InfoData/DcOutputShift
//     Drive/Inputs/In/nState1 <-> Transmit PDO 1/Status Word
//     Drive/Inputs/In/nState2 <-> Transmit PDO 1/Status Word @bit 8
//     Drive/Inputs/In/nState4 @bit 1 <-> WcState/InputToggle
//     Drive/Inputs/In/nState4 <-> WcState/WcState
//     Drive/Outputs/Out/nCtrl1 <-> Receive PDO 1/Control Word
//     Drive/Outputs/Out/nCtrl2 <-> Receive PDO 1/Control Word @bit 8
//     Drive/Outputs/Out/nDataOut1 <-> Receive PDO 1/Profile Target Position
//     Enc/Inputs/In/nDataIn1 <-> Transmit PDO 1/Position Actual Value
//     Enc/Inputs/In/nDataIn3 <-> Transmit PDO 1/Touch Probe 1 Positive Value
//     Enc/Inputs/In/nDcInputTime <-> InfoData/DcInputShift
//     Enc/Inputs/In/nState4 @bit 1 <-> WcState/InputToggle
//     Enc/Inputs/In/nState4 <-> WcState/WcState
//     Enc/Inputs/In/nState5 <-> Transmit PDO 1/Touch Probe Status
//     Enc/Inputs/In/nState6 <-> Transmit PDO 1/Touch Probe Status @bit 8
//     Enc/Outputs/Out/nCtrl5 <-> Receive PDO 1/Touch Probe Function
//     Enc/Outputs/Out/nCtrl6 <-> Receive PDO 1/Touch Probe Function @bit 8
//   NC-Task 1 SAF/Axes/Axis088_40 P2M1_SCurlingneedleWhirling <-> Device 3 (EtherCAT)/P2M1短卷针旋转[40](CL3C-EC808AC)
//     Drive/Inputs/In/nDcOutputTime <-> InfoData/DcOutputShift
//     Drive/Inputs/In/nState1 <-> Transmit PDO 1/Status Word
//     Drive/Inputs/In/nState2 <-> Transmit PDO 1/Status Word @bit 8
//     Drive/Inputs/In/nState4 @bit 1 <-> WcState/InputToggle
//     Drive/Inputs/In/nState4 <-> WcState/WcState
//     Drive/Outputs/Out/nCtrl1 <-> Receive PDO 1/Control Word
//     Drive/Outputs/Out/nCtrl2 <-> Receive PDO 1/Control Word @bit 8
//     Drive/Outputs/Out/nDataOut1 <-> Receive PDO 1/Profile Target Position
//     Enc/Inputs/In/nDataIn1 <-> Transmit PDO 1/Position Actual Value
//     Enc/Inputs/In/nDataIn3 <-> Transmit PDO 1/Touch Probe 1 Positive Value
//     Enc/Inputs/In/nDcInputTime <-> InfoData/DcInputShift
//     Enc/Inputs/In/nState4 @bit 1 <-> WcState/InputToggle
//     Enc/Inputs/In/nState4 <-> WcState/WcState
//     Enc/Inputs/In/nState5 <-> Transmit PDO 1/Touch Probe Status
//     Enc/Inputs/In/nState6 <-> Transmit PDO 1/Touch Probe Status @bit 8
//     Enc/Outputs/Out/nCtrl5 <-> Receive PDO 1/Touch Probe Function
//     Enc/Outputs/Out/nCtrl6 <-> Receive PDO 1/Touch Probe Function @bit 8
//   NC-Task 1 SAF/Axes/Axis089_41 P2M1_GluingLine <-> Device 3 (EtherCAT)/P2M1侧贴夹平移 [41](InoSV660N)
//     Drive/Inputs/In/nDataIn1 <-> Inputs/Following error actual value
//     Drive/Inputs/In/nDcOutputTime <-> InfoData/DcOutputShift
//     Drive/Inputs/In/nState1 <-> Inputs/Statusword
//     Drive/Inputs/In/nState2 <-> Inputs/Statusword @bit 8
//     Drive/Inputs/In/nState4 @bit 1 <-> WcState/InputToggle
//     Drive/Inputs/In/nState4 <-> WcState/WcState
//     Drive/Outputs/Out/nCtrl1 <-> Outputs/Controlword
//     Drive/Outputs/Out/nCtrl2 <-> Outputs/Controlword @bit 8
//     Drive/Outputs/Out/nDataOut1 <-> Outputs/Target position
//     Enc/Inputs/In/nDataIn1 <-> Inputs/Position actual value
//     Enc/Inputs/In/nDataIn3 <-> Inputs/Touch probe pos1 pos value
//     Enc/Inputs/In/nDataIn5 <-> Inputs/Touch probe pos2 pos value
//     Enc/Inputs/In/nDcInputTime <-> InfoData/DcInputShift
//     Enc/Inputs/In/nState4 @bit 1 <-> WcState/InputToggle
//     Enc/Inputs/In/nState4 <-> WcState/WcState
//     Enc/Inputs/In/nState5 <-> Inputs/Touch probe status
//     Enc/Inputs/In/nState6 <-> Inputs/Touch probe status @bit 8
//     Enc/Outputs/Out/nCtrl5 <-> Outputs/Touch probe function
//     Enc/Outputs/Out/nCtrl6 <-> Outputs/Touch probe function @bit 8
//   NC-Task 1 SAF/Axes/Axis090_42 P2M1_GluingWhirling <-> Device 3 (EtherCAT)/P2M1侧贴夹旋转[42] (InoSV660N)
//     Drive/Inputs/In/nDataIn1 <-> Inputs/Following error actual value
//     Drive/Inputs/In/nDcOutputTime <-> InfoData/DcOutputShift
//     Drive/Inputs/In/nState1 <-> Inputs/Statusword
//     Drive/Inputs/In/nState2 <-> Inputs/Statusword @bit 8
//     Drive/Inputs/In/nState4 @bit 1 <-> WcState/InputToggle
//     Drive/Inputs/In/nState4 <-> WcState/WcState
//     Drive/Outputs/Out/nCtrl1 <-> Outputs/Controlword
//     Drive/Outputs/Out/nCtrl2 <-> Outputs/Controlword @bit 8
//     Drive/Outputs/Out/nDataOut1 <-> Outputs/Target position
//     Enc/Inputs/In/nDataIn1 <-> Inputs/Position actual value
//     Enc/Inputs/In/nDataIn3 <-> Inputs/Touch probe pos1 pos value
//     Enc/Inputs/In/nDataIn5 <-> Inputs/Touch probe pos2 pos value
//     Enc/Inputs/In/nDcInputTime <-> InfoData/DcInputShift
//     Enc/Inputs/In/nState4 @bit 1 <-> WcState/InputToggle
//     Enc/Inputs/In/nState4 <-> WcState/WcState
//     Enc/Inputs/In/nState5 <-> Inputs/Touch probe status
//     Enc/Inputs/In/nState6 <-> Inputs/Touch probe status @bit 8
//     Enc/Outputs/Out/nCtrl5 <-> Outputs/Touch probe function
//     Enc/Outputs/Out/nCtrl6 <-> Outputs/Touch probe function @bit 8
//   NC-Task 1 SAF/Axes/Axis091_43 P2M1_GluingRetracting <-> Device 3 (EtherCAT)/P2M1贴胶头进退[43] (InoSV660N)
//     Drive/Inputs/In/nDataIn1 <-> Inputs/Following error actual value
//     Drive/Inputs/In/nDcOutputTime <-> InfoData/DcOutputShift
//     Drive/Inputs/In/nState1 <-> Inputs/Statusword
//     Drive/Inputs/In/nState2 <-> Inputs/Statusword @bit 8
//     Drive/Inputs/In/nState4 @bit 1 <-> WcState/InputToggle
//     Drive/Inputs/In/nState4 <-> WcState/WcState
//     Drive/Outputs/Out/nCtrl1 <-> Outputs/Controlword
//     Drive/Outputs/Out/nCtrl2 <-> Outputs/Controlword @bit 8
//     Drive/Outputs/Out/nDataOut1 <-> Outputs/Target position
//     Enc/Inputs/In/nDataIn1 <-> Inputs/Position actual value
//     Enc/Inputs/In/nDataIn3 <-> Inputs/Touch probe pos1 pos value
//     Enc/Inputs/In/nDataIn5 <-> Inputs/Touch probe pos2 pos value
//     Enc/Inputs/In/nDcInputTime <-> InfoData/DcInputShift
//     Enc/Inputs/In/nState4 @bit 1 <-> WcState/InputToggle
//     Enc/Inputs/In/nState4 <-> WcState/WcState
//     Enc/Inputs/In/nState5 <-> Inputs/Touch probe status
//     Enc/Inputs/In/nState6 <-> Inputs/Touch probe status @bit 8
//     Enc/Outputs/Out/nCtrl5 <-> Outputs/Touch probe function
//     Enc/Outputs/Out/nCtrl6 <-> Outputs/Touch probe function @bit 8
//   NC-Task 1 SAF/Axes/Axis092_44 P2M1_GluingUpDown <-> Device 3 (EtherCAT)/P2M1拉胶升降[44] (InoSV660N)
//     Drive/Inputs/In/nDataIn1 <-> Inputs/Following error actual value
//     Drive/Inputs/In/nDcOutputTime <-> InfoData/DcOutputShift
//     Drive/Inputs/In/nState1 <-> Inputs/Statusword
//     Drive/Inputs/In/nState2 <-> Inputs/Statusword @bit 8
//     Drive/Inputs/In/nState4 @bit 1 <-> WcState/InputToggle
//     Drive/Inputs/In/nState4 <-> WcState/WcState
//     Drive/Outputs/Out/nCtrl1 <-> Outputs/Controlword
//     Drive/Outputs/Out/nCtrl2 <-> Outputs/Controlword @bit 8
//     Drive/Outputs/Out/nDataOut1 <-> Outputs/Target position
//     Enc/Inputs/In/nDataIn1 <-> Inputs/Position actual value
//     Enc/Inputs/In/nDataIn3 <-> Inputs/Touch probe pos1 pos value
//     Enc/Inputs/In/nDataIn5 <-> Inputs/Touch probe pos2 pos value
//     Enc/Inputs/In/nDcInputTime <-> InfoData/DcInputShift
//     Enc/Inputs/In/nState4 @bit 1 <-> WcState/InputToggle
//     Enc/Inputs/In/nState4 <-> WcState/WcState
//     Enc/Inputs/In/nState5 <-> Inputs/Touch probe status
//     Enc/Inputs/In/nState6 <-> Inputs/Touch probe status @bit 8
//     Enc/Outputs/Out/nCtrl5 <-> Outputs/Touch probe function
//     Enc/Outputs/Out/nCtrl6 <-> Outputs/Touch probe function @bit 8
//   NC-Task 1 SAF/Axes/Axis095_47 P2M2_AnCarryingLine <-> Device 3 (EtherCAT)/Box 2 (CU1128)/Term 44 (CU1128-C)/P2M2正极送片搬运平移 [47](CDHD)
//     Drive/Inputs/In/nDataIn1 <-> TxPDO 4/Following Error Actual Value
//     Drive/Inputs/In/nDcOutputTime <-> InfoData/DcOutputShift
//     Drive/Inputs/In/nState1 <-> TxPDO 1/StatusWord
//     Drive/Inputs/In/nState2 <-> TxPDO 1/StatusWord @bit 8
//     Drive/Inputs/In/nState4 @bit 1 <-> WcState/InputToggle
//     Drive/Inputs/In/nState4 <-> WcState/WcState
//     Drive/Inputs/In/nState5 <-> TxPDO 1/Modes of operation display
//     Drive/Outputs/Out/nCtrl1 <-> RxPDO 1/ControlWord
//     Drive/Outputs/Out/nCtrl2 <-> RxPDO 1/ControlWord @bit 8
//     Drive/Outputs/Out/nCtrl5 <-> RxPDO 1/Modes of operation
//     Drive/Outputs/Out/nDataOut1 <-> RxPDO 2/Target position
//     Drive/Outputs/Out/nDataOut2 <-> RxPDO 3/Target Velocity
//     Drive/Outputs/Out/nDataOut3[0] <-> RxPDO 4/Torque Offset
//     Drive/Outputs/Out/nDataOut4[0] <-> RxPDO 4/Target torque
//     Enc/Inputs/In/nDataIn1 <-> TxPDO 2/Position actual value
//     Enc/Inputs/In/nDcInputTime <-> InfoData/DcInputShift
//     Enc/Inputs/In/nState4 @bit 1 <-> WcState/InputToggle
//     Enc/Inputs/In/nState4 <-> WcState/WcState
//   NC-Task 1 SAF/Axes/Axis096_48 P2M2_AnCarryingUpDown <-> Device 3 (EtherCAT)/Box 2 (CU1128)/Term 44 (CU1128-C)/P2M2正极送片搬运升降[48] (InoSV660N)
//     Drive/Inputs/In/nDataIn1 <-> Inputs/Following error actual value
//     Drive/Inputs/In/nDcOutputTime <-> InfoData/DcOutputShift
//     Drive/Inputs/In/nState1 <-> Inputs/Statusword
//     Drive/Inputs/In/nState2 <-> Inputs/Statusword @bit 8
//     Drive/Inputs/In/nState4 @bit 1 <-> WcState/InputToggle
//     Drive/Inputs/In/nState4 <-> WcState/WcState
//     Drive/Outputs/Out/nCtrl1 <-> Outputs/Controlword
//     Drive/Outputs/Out/nCtrl2 <-> Outputs/Controlword @bit 8
//     Drive/Outputs/Out/nDataOut1 <-> Outputs/Target position
//     Enc/Inputs/In/nDataIn1 <-> Inputs/Position actual value
//     Enc/Inputs/In/nDataIn3 <-> Inputs/Touch probe pos1 pos value
//     Enc/Inputs/In/nDataIn5 <-> Inputs/Touch probe pos2 pos value
//     Enc/Inputs/In/nDcInputTime <-> InfoData/DcInputShift
//     Enc/Inputs/In/nState4 @bit 1 <-> WcState/InputToggle
//     Enc/Inputs/In/nState4 <-> WcState/WcState
//     Enc/Inputs/In/nState5 <-> Inputs/Touch probe status
//     Enc/Inputs/In/nState6 <-> Inputs/Touch probe status @bit 8
//     Enc/Outputs/Out/nCtrl5 <-> Outputs/Touch probe function
//     Enc/Outputs/Out/nCtrl6 <-> Outputs/Touch probe function @bit 8
//   NC-Task 1 SAF/Axes/Axis097_49 P2M2_AnCarryingWhirling <-> Device 3 (EtherCAT)/Box 2 (CU1128)/Term 44 (CU1128-C)/P2M2正极送片搬运旋转[49] (InoSV660N)
//     Drive/Inputs/In/nDataIn1 <-> Inputs/Following error actual value
//     Drive/Inputs/In/nDcOutputTime <-> InfoData/DcOutputShift
//     Drive/Inputs/In/nState1 <-> Inputs/Statusword
//     Drive/Inputs/In/nState2 <-> Inputs/Statusword @bit 8
//     Drive/Inputs/In/nState4 @bit 1 <-> WcState/InputToggle
//     Drive/Inputs/In/nState4 <-> WcState/WcState
//     Drive/Outputs/Out/nCtrl1 <-> Outputs/Controlword
//     Drive/Outputs/Out/nCtrl2 <-> Outputs/Controlword @bit 8
//     Drive/Outputs/Out/nDataOut1 <-> Outputs/Target position
//     Enc/Inputs/In/nDataIn1 <-> Inputs/Position actual value
//     Enc/Inputs/In/nDataIn3 <-> Inputs/Touch probe pos1 pos value
//     Enc/Inputs/In/nDataIn5 <-> Inputs/Touch probe pos2 pos value
//     Enc/Inputs/In/nDcInputTime <-> InfoData/DcInputShift
//     Enc/Inputs/In/nState4 @bit 1 <-> WcState/InputToggle
//     Enc/Inputs/In/nState4 <-> WcState/WcState
//     Enc/Inputs/In/nState5 <-> Inputs/Touch probe status
//     Enc/Inputs/In/nState6 <-> Inputs/Touch probe status @bit 8
//     Enc/Outputs/Out/nCtrl5 <-> Outputs/Touch probe function
//     Enc/Outputs/Out/nCtrl6 <-> Outputs/Touch probe function @bit 8
//   NC-Task 1 SAF/Axes/Axis098_50 P2M2_AnDTCarryingLine <-> Device 3 (EtherCAT)/Box 2 (CU1128)/Term 44 (CU1128-C)/P2M2正极叠台搬运平移1[50](CDHD)
//     Drive/Inputs/In/nDataIn1 <-> TxPDO 4/Following Error Actual Value
//     Drive/Inputs/In/nDcOutputTime <-> InfoData/DcOutputShift
//     Drive/Inputs/In/nState1 <-> TxPDO 1/StatusWord
//     Drive/Inputs/In/nState2 <-> TxPDO 1/StatusWord @bit 8
//     Drive/Inputs/In/nState4 @bit 1 <-> WcState/InputToggle
//     Drive/Inputs/In/nState4 <-> WcState/WcState
//     Drive/Inputs/In/nState5 <-> TxPDO 1/Modes of operation display
//     Drive/Outputs/Out/nCtrl1 <-> RxPDO 1/ControlWord
//     Drive/Outputs/Out/nCtrl2 <-> RxPDO 1/ControlWord @bit 8
//     Drive/Outputs/Out/nCtrl5 <-> RxPDO 1/Modes of operation
//     Drive/Outputs/Out/nDataOut1 <-> RxPDO 2/Target position
//     Drive/Outputs/Out/nDataOut2 <-> RxPDO 3/Target Velocity
//     Drive/Outputs/Out/nDataOut3[0] <-> RxPDO 4/Torque Offset
//     Drive/Outputs/Out/nDataOut4[0] <-> RxPDO 4/Target torque
//     Enc/Inputs/In/nDataIn1 <-> TxPDO 2/Position actual value
//     Enc/Inputs/In/nDcInputTime <-> InfoData/DcInputShift
//     Enc/Inputs/In/nState4 @bit 1 <-> WcState/InputToggle
//     Enc/Inputs/In/nState4 <-> WcState/WcState
//   NC-Task 1 SAF/Axes/Axis099_51 P2M2_AnDTCarryingUpDown <-> Device 3 (EtherCAT)/Box 2 (CU1128)/Term 44 (CU1128-C)/P2M2正极叠台搬运升降[51] (InoSV660N)
//     Drive/Inputs/In/nDataIn1 <-> Inputs/Following error actual value
//     Drive/Inputs/In/nDcOutputTime <-> InfoData/DcOutputShift
//     Drive/Inputs/In/nState1 <-> Inputs/Statusword
//     Drive/Inputs/In/nState2 <-> Inputs/Statusword @bit 8
//     Drive/Inputs/In/nState4 @bit 1 <-> WcState/InputToggle
//     Drive/Inputs/In/nState4 <-> WcState/WcState
//     Drive/Outputs/Out/nCtrl1 <-> Outputs/Controlword
//     Drive/Outputs/Out/nCtrl2 <-> Outputs/Controlword @bit 8
//     Drive/Outputs/Out/nDataOut1 <-> Outputs/Target position
//     Enc/Inputs/In/nDataIn1 <-> Inputs/Position actual value
//     Enc/Inputs/In/nDataIn3 <-> Inputs/Touch probe pos1 pos value
//     Enc/Inputs/In/nDataIn5 <-> Inputs/Touch probe pos2 pos value
//     Enc/Inputs/In/nDcInputTime <-> InfoData/DcInputShift
//     Enc/Inputs/In/nState4 @bit 1 <-> WcState/InputToggle
//     Enc/Inputs/In/nState4 <-> WcState/WcState
//     Enc/Inputs/In/nState5 <-> Inputs/Touch probe status
//     Enc/Inputs/In/nState6 <-> Inputs/Touch probe status @bit 8
//     Enc/Outputs/Out/nCtrl5 <-> Outputs/Touch probe function
//     Enc/Outputs/Out/nCtrl6 <-> Outputs/Touch probe function @bit 8
//   NC-Task 1 SAF/Axes/Axis100_52 P2M2_AndeviationX1 <-> Device 3 (EtherCAT)/Box 2 (CU1128)/Term 44 (CU1128-C)/P2M2正极纠偏平台X1[52] (InoSV660N)
//     Drive/Inputs/In/nDataIn1 <-> Inputs/Following error actual value
//     Drive/Inputs/In/nDcOutputTime <-> InfoData/DcOutputShift
//     Drive/Inputs/In/nState1 <-> Inputs/Statusword
//     Drive/Inputs/In/nState2 <-> Inputs/Statusword @bit 8
//     Drive/Inputs/In/nState4 @bit 1 <-> WcState/InputToggle
//     Drive/Inputs/In/nState4 <-> WcState/WcState
//     Drive/Outputs/Out/nCtrl1 <-> Outputs/Controlword
